LIN {X 0,Y 144.204,Z 524.14,A -85,B 0,C 180,E1 -26321.99,E2 -26321.99} C_VEL
LIN {X 0,Y 135.871,Z 530.336,A -85,B 0,C 180,E1 -26325.708,E2 -26325.708} C_VEL
LIN {X 0,Y 129.15,Z 534.492,A -85,B 0,C 180,E1 -26329.229,E2 -26329.229} C_VEL
LIN {X 0,Y 124.469,Z 537.046,A -85,B 0,C 180,E1 -26332.231,E2 -26332.231} C_VEL
LIN {X 0,Y 117.932,Z 540.01,A -85,B 0,C 180,E1 -26337.563,E2 -26337.563} C_VEL
LIN {X 0,Y 112.138,Z 541.802,A -85,B 0,C 180,E1 -26343.976,E2 -26343.976} C_VEL
LIN {X 0,Y 108.067,Z 542.166,A -85,B 0,C 180,E1 -26351.022,E2 -26351.022} C_VEL
LIN {X 0,Y 105.891,Z 541.033,A -85,B 0,C 180,E1 -26358.513,E2 -26358.513} C_VEL
LIN {X 0,Y 105.433,Z 538.416,A -85,B 0,C 180,E1 -26366.176,E2 -26366.176} C_VEL
LIN {X 0,Y 105.739,Z 536.5,A -85,B 0,C 180,E1 -26369.998,E2 -26369.998} C_VEL
LIN {X 0,Y 105.585,Z 532.557,A -85,B 0,C 180,E1 -26375.728,E2 -26375.728} C_VEL
LIN {X 0,Y 106.291,Z 526.365,A -85,B 0,C 180,E1 -26382.407,E2 -26382.407} C_VEL
LIN {X 0,Y 107.726,Z 519.519,A -85,B 0,C 180,E1 -26388.05,E2 -26388.05} C_VEL
LIN {X 0,Y 110.21,Z 510.988,A -85,B 0,C 180,E1 -26393.485,E2 -26393.485} C_VEL
LIN {X 0,Y 112.838,Z 502.152,A -85,B 0,C 180,E1 -26397.845,E2 -26397.845} C_VEL
LIN {X 0,Y 115.825,Z 492.148,A -85,B 0,C 180,E1 -26401.702,E2 -26401.702} C_VEL
LIN {X 0,Y 118.812,Z 482.066,A -85,B 0,C 180,E1 -26404.702,E2 -26404.702} C_VEL
LIN {X 0,Y 121.726,Z 470.618,A -85,B 0,C 180,E1 -26407.315,E2 -26407.315} C_VEL
LIN {X 0,Y 123.606,Z 461.97,A -85,B 0,C 180,E1 -26408.845,E2 -26408.845} C_VEL
LIN {X 0,Y 123.986,Z 456.45,A -85,B 0,C 180,E1 -26409.818,E2 -26409.818} C_VEL
LIN {X 0,Y 122.886,Z 447.257,A -85,B 0,C 180,E1 -26411.482,E2 -26411.482} C_VEL
LIN {X 0,Y 121.565,Z 437.876,A -85,B 0,C 180,E1 -26412.9,E2 -26412.9} C_VEL
LIN {X 0,Y 121.526,Z 432.057,A -85,B 0,C 180,E1 -26413.443,E2 -26413.443} C_VEL
LIN {X 0,Y 124.402,Z 398.174,A -85,B 0,C 180,E1 -26415.575,E2 -26415.575} C_VEL
LIN {X 0,Y 123.704,Z 390.073,A -85,B 0,C 180,E1 -26416.461,E2 -26416.461} C_VEL
LIN {X 0,Y 118.365,Z 373.234,A -85,B 0,C 180,E1 -26419.573,E2 -26419.573} C_VEL
LIN {X 0,Y 113.624,Z 360.938,A -85,B 0,C 180,E1 -26422.379,E2 -26422.379} C_VEL
LIN {X 0,Y 107.274,Z 349.28,A -85,B 0,C 180,E1 -26426.161,E2 -26426.161} C_VEL
LIN {X 0,Y 104.542,Z 345.011,A -85,B 0,C 180,E1 -26427.85,E2 -26427.85} C_VEL
LIN {X 0,Y 102.828,Z 342.099,A -85,B 0,C 180,E1 -26429.006,E2 -26429.006} C_VEL
LIN {X 0,Y 101.238,Z 339.918,A -85,B 0,C 180,E1 -26430.07,E2 -26430.07} C_VEL
LIN {X 0,Y 100.677,Z 337.944,A -85,B 0,C 180,E1 -26430.606,E2 -26430.606} C_VEL
LIN {X 0,Y 100.782,Z 337.935,A -85,B 0,C 180,E1 -26435.267,E2 -26435.267} C_VEL
LIN {X 0,Y 100.814,Z 337.916,A -85,B 0,C 180,E1 -26439.601,E2 -26439.601} C_VEL
LIN {X 0,Y 101.184,Z 337.863,A -85,B 0,C 180,E1 -26447.974,E2 -26447.974} C_VEL
LIN {X 0,Y 101.264,Z 337.87,A -85,B 0,C 180,E1 -26452.022,E2 -26452.022} C_VEL
LIN {X 0,Y 101.841,Z 337.774,A -85,B 0,C 180,E1 -26460.001,E2 -26460.001} C_VEL
LIN {X 0,Y 101.237,Z 337.86,A -85,B 0,C 180,E1 -26467.982,E2 -26467.982} C_VEL
LIN {X 0,Y 101.1,Z 337.863,A -85,B 0,C 180,E1 -26473.303,E2 -26473.303} C_VEL
LIN {X 0,Y 100.812,Z 337.919,A -85,B 0,C 180,E1 -26480.401,E2 -26480.401} C_VEL
LIN {X 0,Y 100.771,Z 337.896,A -85,B 0,C 180,E1 -26484.961,E2 -26484.961} C_VEL
LIN {X 0,Y 100.685,Z 337.943,A -85,B 0,C 180,E1 -26493.115,E2 -26493.115} C_VEL
LIN {X 0,Y 100.633,Z 337.918,A -85,B 0,C 180,E1 -26499.81,E2 -26499.81} C_VEL
LIN {X 0,Y 100.639,Z 337.948,A -85,B 0,C 180,E1 -26505.71,E2 -26505.71} C_VEL
LIN {X 0,Y 100.619,Z 337.931,A -85,B 0,C 180,E1 -26511.054,E2 -26511.054} C_VEL
LIN {X 0,Y 100.687,Z 337.941,A -85,B 0,C 180,E1 -26516.89,E2 -26516.89} C_VEL
LIN {X 0,Y 100.787,Z 337.927,A -85,B 0,C 180,E1 -26525.27,E2 -26525.27} C_VEL
LIN {X 0,Y 100.805,Z 337.924,A -85,B 0,C 180,E1 -26529.601,E2 -26529.601} C_VEL
LIN {X 0,Y 101.125,Z 337.885,A -85,B 0,C 180,E1 -26537.331,E2 -26537.331} C_VEL
LIN {X 0,Y 102.17,Z 340.771,A -85,B 0,C 180,E1 -26538.28,E2 -26538.28} C_VEL
LIN {X 0,Y 104.082,Z 343.292,A -85,B 0,C 180,E1 -26539.517,E2 -26539.517} C_VEL
LIN {X 0,Y 112.366,Z 356.593,A -85,B 0,C 180,E1 -26544.485,E2 -26544.485} C_VEL
LIN {X 0,Y 119.927,Z 373.331,A -85,B 0,C 180,E1 -26548.715,E2 -26548.715} C_VEL
LIN {X 0,Y 124.992,Z 386.089,A -85,B 0,C 180,E1 -26551.329,E2 -26551.329} C_VEL
LIN {X 0,Y 121.055,Z 431.333,A -85,B 0,C 180,E1 -26554.206,E2 -26554.206} C_VEL
LIN {X 0,Y 119.221,Z 444.562,A -85,B 0,C 180,E1 -26555.591,E2 -26555.591} C_VEL
LIN {X 0,Y 116.791,Z 457.435,A -85,B 0,C 180,E1 -26557.566,E2 -26557.566} C_VEL
LIN {X 0,Y 113.893,Z 469.698,A -85,B 0,C 180,E1 -26560.203,E2 -26560.203} C_VEL
LIN {X 0,Y 110.823,Z 480.586,A -85,B 0,C 180,E1 -26563.292,E2 -26563.292} C_VEL
LIN {X 0,Y 107.694,Z 490.863,A -85,B 0,C 180,E1 -26567.078,E2 -26567.078} C_VEL
LIN {X 0,Y 104.784,Z 499.838,A -85,B 0,C 180,E1 -26571.312,E2 -26571.312} C_VEL
LIN {X 0,Y 102.059,Z 508.347,A -85,B 0,C 180,E1 -26576.462,E2 -26576.462} C_VEL
LIN {X 0,Y 99.906,Z 516.005,A -85,B 0,C 180,E1 -26582.416,E2 -26582.416} C_VEL
LIN {X 0,Y 98.446,Z 521.87,A -85,B 0,C 180,E1 -26588.251,E2 -26588.251} C_VEL
LIN {X 0,Y 97.658,Z 526.395,A -85,B 0,C 180,E1 -26593.972,E2 -26593.972} C_VEL
LIN {X 0,Y 97.689,Z 529.93,A -85,B 0,C 180,E1 -26599.646,E2 -26599.646} C_VEL
LIN {X 0,Y 98.406,Z 532.573,A -85,B 0,C 180,E1 -26605.154,E2 -26605.154} C_VEL
LIN {X 0,Y 99.872,Z 534.421,A -85,B 0,C 180,E1 -26610.488,E2 -26610.488} C_VEL
LIN {X 0,Y 102.065,Z 535.611,A -85,B 0,C 180,E1 -26615.596,E2 -26615.596} C_VEL
LIN {X 0,Y 104.928,Z 536.153,A -85,B 0,C 180,E1 -26620.433,E2 -26620.433} C_VEL
LIN {X 0,Y 108.909,Z 535.995,A -85,B 0,C 180,E1 -26625.465,E2 -26625.465} C_VEL
LIN {X 0,Y 114.037,Z 534.986,A -85,B 0,C 180,E1 -26630.435,E2 -26630.435} C_VEL
LIN {X 0,Y 119.949,Z 533.081,A -85,B 0,C 180,E1 -26634.927,E2 -26634.927} C_VEL
LIN {X 0,Y 128.424,Z 529.271,A -85,B 0,C 180,E1 -26639.999,E2 -26639.999} C_VEL
LIN {X 0,Y 136.2,Z 524.843,A -85,B 0,C 180,E1 -26643.698,E2 -26643.698} C_VEL
LIN {X 0,Y 144.662,Z 519.043,A -85,B 0,C 180,E1 -26646.994,E2 -26646.994} C_VEL
LIN {X 0,Y 152.275,Z 512.818,A -85,B 0,C 180,E1 -26649.517,E2 -26649.517} C_VEL
LIN {X 0,Y 160.205,Z 505.173,A -85,B 0,C 180,E1 -26651.777,E2 -26651.777} C_VEL
LIN {X 0,Y 168.345,Z 495.926,A -85,B 0,C 180,E1 -26653.794,E2 -26653.794} C_VEL
LIN {X 0,Y 175.893,Z 485.667,A -85,B 0,C 180,E1 -26655.433,E2 -26655.433} C_VEL
LIN {X 0,Y 182.758,Z 474.132,A -85,B 0,C 180,E1 -26656.795,E2 -26656.795} C_VEL
LIN {X 0,Y 188.597,Z 461.804,A -85,B 0,C 180,E1 -26657.91,E2 -26657.91} C_VEL
LIN {X 0,Y 192.89,Z 449.978,A -85,B 0,C 180,E1 -26658.678,E2 -26658.678} C_VEL
LIN {X 0,Y 195.848,Z 439.157,A -85,B 0,C 180,E1 -26659.203,E2 -26659.203} C_VEL
LIN {X 0,Y 195.57,Z 437.962,A -85,B 0,C 180,E1 -26662.113,E2 -26662.113} C_VEL
LIN {X 0,Y 195.496,Z 438.41,A -85,B 0,C 180,E1 -26664.285,E2 -26664.285} C_VEL
LIN {X 0,Y 195.538,Z 441.194,A -85,B 0,C 180,E1 -26667.429,E2 -26667.429} C_VEL
LIN {X 0,Y 191.453,Z 455.147,A -85,B 0,C 180,E1 -26667.987,E2 -26667.987} C_VEL
LIN {X 0,Y 186.227,Z 468.207,A -85,B 0,C 180,E1 -26668.756,E2 -26668.756} C_VEL
LIN {X 0,Y 180.077,Z 480.052,A -85,B 0,C 180,E1 -26669.729,E2 -26669.729} C_VEL
LIN {X 0,Y 173.13,Z 490.968,A -85,B 0,C 180,E1 -26670.956,E2 -26670.956} C_VEL
LIN {X 0,Y 166.328,Z 499.92,A -85,B 0,C 180,E1 -26672.318,E2 -26672.318} C_VEL
LIN {X 0,Y 157.53,Z 509.729,A -85,B 0,C 180,E1 -26674.374,E2 -26674.374} C_VEL
LIN {X 0,Y 149.078,Z 517.709,A -85,B 0,C 180,E1 -26676.731,E2 -26676.731} C_VEL
LIN {X 0,Y 140.938,Z 524.241,A -85,B 0,C 180,E1 -26679.381,E2 -26679.381} C_VEL
LIN {X 0,Y 133.327,Z 529.522,A -85,B 0,C 180,E1 -26682.439,E2 -26682.439} C_VEL
LIN {X 0,Y 126.142,Z 533.783,A -85,B 0,C 180,E1 -26685.856,E2 -26685.856} C_VEL
LIN {X 0,Y 118.487,Z 537.566,A -85,B 0,C 180,E1 -26690.451,E2 -26690.451} C_VEL
LIN {X 0,Y 112.005,Z 540.093,A -85,B 0,C 180,E1 -26695.615,E2 -26695.615} C_VEL
LIN {X 0,Y 105.797,Z 541.664,A -85,B 0,C 180,E1 -26702.287,E2 -26702.287} C_VEL
LIN {X 0,Y 101.349,Z 541.752,A -85,B 0,C 180,E1 -26709.711,E2 -26709.711} C_VEL
LIN {X 0,Y 98.949,Z 540.44,A -85,B 0,C 180,E1 -26717.695,E2 -26717.695} C_VEL
LIN {X 0,Y 98.445,Z 539.235,A -85,B 0,C 180,E1 -26721.789,E2 -26721.789} C_VEL
LIN {X 0,Y 98.499,Z 536.938,A -85,B 0,C 180,E1 -26727.315,E2 -26727.315} C_VEL
LIN {X 0,Y 98.683,Z 535.535,A -85,B 0,C 180,E1 -26729.998,E2 -26729.998} C_VEL
LIN {X 0,Y 98.543,Z 531.382,A -85,B 0,C 180,E1 -26736.139,E2 -26736.139} C_VEL
LIN {X 0,Y 99.189,Z 525.985,A -85,B 0,C 180,E1 -26742.27,E2 -26742.27} C_VEL
LIN {X 0,Y 100.645,Z 519.146,A -85,B 0,C 180,E1 -26748.312,E2 -26748.312} C_VEL
LIN {X 0,Y 103.205,Z 510.618,A -85,B 0,C 180,E1 -26754.113,E2 -26754.113} C_VEL
LIN {X 0,Y 105.951,Z 501.798,A -85,B 0,C 180,E1 -26758.742,E2 -26758.742} C_VEL
LIN {X 0,Y 109.22,Z 491.411,A -85,B 0,C 180,E1 -26762.954,E2 -26762.954} C_VEL
LIN {X 0,Y 112.206,Z 481.72,A -85,B 0,C 180,E1 -26765.956,E2 -26765.956} C_VEL
LIN {X 0,Y 115.243,Z 470.241,A -85,B 0,C 180,E1 -26768.686,E2 -26768.686} C_VEL
LIN {X 0,Y 118.067,Z 457.449,A -85,B 0,C 180,E1 -26770.9,E2 -26770.9} C_VEL
LIN {X 0,Y 120.301,Z 444.156,A -85,B 0,C 180,E1 -26772.489,E2 -26772.489} C_VEL
LIN {X 0,Y 121.526,Z 432.057,A -85,B 0,C 180,E1 -26773.443,E2 -26773.443} C_VEL
LIN {X 0,Y 121.435,Z 426.244,A -85,B 0,C 180,E1 -26773.965,E2 -26773.965} C_VEL
LIN {X 0,Y 118.145,Z 407.407,A -85,B 0,C 180,E1 -26776.532,E2 -26776.532} C_VEL
LIN {X 0,Y 118.126,Z 401.597,A -85,B 0,C 180,E1 -26777.059,E2 -26777.059} C_VEL
LIN {X 0,Y 118.078,Z 394.458,A -85,B 0,C 180,E1 -26777.721,E2 -26777.721} C_VEL
LIN {X 0,Y 117.409,Z 390.896,A -85,B 0,C 180,E1 -26778.246,E2 -26778.246} C_VEL
LIN {X 0,Y 112.107,Z 374.256,A -85,B 0,C 180,E1 -26781.6,E2 -26781.6} C_VEL
LIN {X 0,Y 108.138,Z 364.014,A -85,B 0,C 180,E1 -26784.203,E2 -26784.203} C_VEL
LIN {X 0,Y 101.886,Z 352.501,A -85,B 0,C 180,E1 -26788.245,E2 -26788.245} C_VEL
LIN {X 0,Y 98.227,Z 346.757,A -85,B 0,C 180,E1 -26790.829,E2 -26790.829} C_VEL
LIN {X 0,Y 96.222,Z 343.476,A -85,B 0,C 180,E1 -26792.398,E2 -26792.398} C_VEL
LIN {X 0,Y 94.338,Z 341.074,A -85,B 0,C 180,E1 -26793.879,E2 -26793.879} C_VEL
LIN {X 0,Y 93.705,Z 338.814,A -85,B 0,C 180,E1 -26794.634,E2 -26794.634} C_VEL
LIN {X 0,Y 93.789,Z 338.802,A -85,B 0,C 180,E1 -26802.559,E2 -26802.559} C_VEL
LIN {X 0,Y 94.088,Z 338.749,A -85,B 0,C 180,E1 -26807.052,E2 -26807.052} C_VEL
LIN {X 0,Y 94.197,Z 338.747,A -85,B 0,C 180,E1 -26811.419,E2 -26811.419} C_VEL
LIN {X 0,Y 94.77,Z 338.654,A -85,B 0,C 180,E1 -26820.001,E2 -26820.001} C_VEL
LIN {X 0,Y 94.171,Z 338.734,A -85,B 0,C 180,E1 -26828.585,E2 -26828.585} C_VEL
LIN {X 0,Y 94.02,Z 338.745,A -85,B 0,C 180,E1 -26833.663,E2 -26833.663} C_VEL
LIN {X 0,Y 93.689,Z 338.797,A -85,B 0,C 180,E1 -26842.03,E2 -26842.03} C_VEL
LIN {X 0,Y 93.616,Z 338.789,A -85,B 0,C 180,E1 -26846.773,E2 -26846.773} C_VEL
LIN {X 0,Y 93.582,Z 338.826,A -85,B 0,C 180,E1 -26854.305,E2 -26854.305} C_VEL
LIN {X 0,Y 93.526,Z 338.814,A -85,B 0,C 180,E1 -26862.557,E2 -26862.557} C_VEL
LIN {X 0,Y 93.529,Z 338.829,A -85,B 0,C 180,E1 -26868.716,E2 -26868.716} C_VEL
LIN {X 0,Y 93.583,Z 338.819,A -85,B 0,C 180,E1 -26875.702,E2 -26875.702} C_VEL
LIN {X 0,Y 93.668,Z 338.816,A -85,B 0,C 180,E1 -26884.209,E2 -26884.209} C_VEL
LIN {X 0,Y 93.687,Z 338.814,A -85,B 0,C 180,E1 -26887.974,E2 -26887.974} C_VEL
LIN {X 0,Y 93.799,Z 338.942,A -85,B 0,C 180,E1 -26893.278,E2 -26893.278} C_VEL
LIN {X 0,Y 94.891,Z 341.725,A -85,B 0,C 180,E1 -26894.334,E2 -26894.334} C_VEL
LIN {X 0,Y 97.123,Z 344.099,A -85,B 0,C 180,E1 -26895.967,E2 -26895.967} C_VEL
LIN {X 0,Y 99.179,Z 347.343,A -85,B 0,C 180,E1 -26897.528,E2 -26897.528} C_VEL
LIN {X 0,Y 107.498,Z 360.915,A -85,B 0,C 180,E1 -26902.987,E2 -26902.987} C_VEL
LIN {X 0,Y 114.636,Z 377.165,A -85,B 0,C 180,E1 -26907.352,E2 -26907.352} C_VEL
LIN {X 0,Y 118.889,Z 388.434,A -85,B 0,C 180,E1 -26909.767,E2 -26909.767} C_VEL
LIN {X 0,Y 114.656,Z 432.343,A -85,B 0,C 180,E1 -26912.641,E2 -26912.641} C_VEL
LIN {X 0,Y 112.746,Z 445.688,A -85,B 0,C 180,E1 -26914.15,E2 -26914.15} C_VEL
LIN {X 0,Y 110.205,Z 458.188,A -85,B 0,C 180,E1 -26916.178,E2 -26916.178} C_VEL
LIN {X 0,Y 107.152,Z 470.365,A -85,B 0,C 180,E1 -26918.945,E2 -26918.945} C_VEL
LIN {X 0,Y 104.007,Z 481.143,A -85,B 0,C 180,E1 -26922.192,E2 -26922.192} C_VEL
LIN {X 0,Y 100.671,Z 491.438,A -85,B 0,C 180,E1 -26926.218,E2 -26926.218} C_VEL
LIN {X 0,Y 97.377,Z 501.07,A -85,B 0,C 180,E1 -26931.156,E2 -26931.156} C_VEL
LIN {X 0,Y 94.561,Z 509.672,A -85,B 0,C 180,E1 -26936.887,E2 -26936.887} C_VEL
LIN {X 0,Y 92.485,Z 517.112,A -85,B 0,C 180,E1 -26943.288,E2 -26943.288} C_VEL
LIN {X 0,Y 91.086,Z 522.715,A -85,B 0,C 180,E1 -26949.502,E2 -26949.502} C_VEL
LIN {X 0,Y 90.487,Z 527.069,A -85,B 0,C 180,E1 -26955.65,E2 -26955.65} C_VEL
LIN {X 0,Y 90.756,Z 530.464,A -85,B 0,C 180,E1 -26961.718,E2 -26961.718} C_VEL
LIN {X 0,Y 91.8,Z 533.031,A -85,B 0,C 180,E1 -26967.593,E2 -26967.593} C_VEL
LIN {X 0,Y 93.916,Z 535.029,A -85,B 0,C 180,E1 -26973.9,E2 -26973.9} C_VEL
LIN {X 0,Y 97.161,Z 536.19,A -85,B 0,C 180,E1 -26980.113,E2 -26980.113} C_VEL
LIN {X 0,Y 101.446,Z 536.477,A -85,B 0,C 180,E1 -26985.914,E2 -26985.914} C_VEL
LIN {X 0,Y 108.249,Z 535.606,A -85,B 0,C 180,E1 -26992.538,E2 -26992.538} C_VEL
LIN {X 0,Y 116.34,Z 533.242,A -85,B 0,C 180,E1 -26998.268,E2 -26998.268} C_VEL
LIN {X 0,Y 125.407,Z 529.439,A -85,B 0,C 180,E1 -27003.212,E2 -27003.212} C_VEL
LIN {X 0,Y 134.561,Z 524.463,A -85,B 0,C 180,E1 -27007.078,E2 -27007.078} C_VEL
LIN {X 0,Y 144.5,Z 517.663,A -85,B 0,C 180,E1 -27010.519,E2 -27010.519} C_VEL
LIN {X 0,Y 153.935,Z 509.908,A -85,B 0,C 180,E1 -27013.195,E2 -27013.195} C_VEL
LIN {X 0,Y 162.792,Z 501.042,A -85,B 0,C 180,E1 -27015.326,E2 -27015.326} C_VEL
LIN {X 0,Y 170.888,Z 491.294,A -85,B 0,C 180,E1 -27017.039,E2 -27017.039} C_VEL
LIN {X 0,Y 178.182,Z 480.655,A -85,B 0,C 180,E1 -27018.393,E2 -27018.393} C_VEL
LIN {X 0,Y 184.909,Z 468.504,A -85,B 0,C 180,E1 -27019.569,E2 -27019.569} C_VEL
LIN {X 0,Y 190.067,Z 456.664,A -85,B 0,C 180,E1 -27020.435,E2 -27020.435} C_VEL
LIN {X 0,Y 193.832,Z 445.249,A -85,B 0,C 180,E1 -27021.052,E2 -27021.052} C_VEL
LIN {X 0,Y 193.728,Z 445.121,A -85,B 0,C 180,E1 -27023.844,E2 -27023.844} C_VEL
LIN {X 0,Y 193.618,Z 445.986,A -85,B 0,C 180,E1 -27024.842,E2 -27024.842} C_VEL
LIN {X 0,Y 193.316,Z 447.422,A -85,B 0,C 180,E1 -27025.56,E2 -27025.56} C_VEL
LIN {X 0,Y 188.554,Z 460.936,A -85,B 0,C 180,E1 -27026.137,E2 -27026.137} C_VEL
LIN {X 0,Y 183.163,Z 472.612,A -85,B 0,C 180,E1 -27026.859,E2 -27026.859} C_VEL
LIN {X 0,Y 175.98,Z 484.888,A -85,B 0,C 180,E1 -27027.919,E2 -27027.919} C_VEL
LIN {X 0,Y 168.914,Z 494.863,A -85,B 0,C 180,E1 -27029.101,E2 -27029.101} C_VEL
LIN {X 0,Y 161.229,Z 503.991,A -85,B 0,C 180,E1 -27030.579,E2 -27030.579} C_VEL
LIN {X 0,Y 152.238,Z 512.942,A -85,B 0,C 180,E1 -27032.592,E2 -27032.592} C_VEL
LIN {X 0,Y 142.182,Z 521.313,A -85,B 0,C 180,E1 -27035.352,E2 -27035.352} C_VEL
LIN {X 0,Y 133.834,Z 527.14,A -85,B 0,C 180,E1 -27038.027,E2 -27038.027} C_VEL
LIN {X 0,Y 126.165,Z 531.775,A -85,B 0,C 180,E1 -27041.233,E2 -27041.233} C_VEL
LIN {X 0,Y 118.795,Z 535.449,A -85,B 0,C 180,E1 -27044.769,E2 -27044.769} C_VEL
LIN {X 0,Y 110.073,Z 538.977,A -85,B 0,C 180,E1 -27050.318,E2 -27050.318} C_VEL
LIN {X 0,Y 102.653,Z 540.981,A -85,B 0,C 180,E1 -27056.787,E2 -27056.787} C_VEL
LIN {X 0,Y 96.842,Z 541.563,A -85,B 0,C 180,E1 -27064.185,E2 -27064.185} C_VEL
LIN {X 0,Y 93.142,Z 540.758,A -85,B 0,C 180,E1 -27072.431,E2 -27072.431} C_VEL
LIN {X 0,Y 91.442,Z 538.447,A -85,B 0,C 180,E1 -27081.155,E2 -27081.155} C_VEL
LIN {X 0,Y 91.465,Z 535.97,A -85,B 0,C 180,E1 -27087.298,E2 -27087.298} C_VEL
LIN {X 0,Y 91.62,Z 534.567,A -85,B 0,C 180,E1 -27089.997,E2 -27089.997} C_VEL
LIN {X 0,Y 91.508,Z 530.203,A -85,B 0,C 180,E1 -27096.613,E2 -27096.613} C_VEL
LIN {X 0,Y 92.254,Z 524.573,A -85,B 0,C 180,E1 -27103.209,E2 -27103.209} C_VEL
LIN {X 0,Y 93.945,Z 517.428,A -85,B 0,C 180,E1 -27109.67,E2 -27109.67} C_VEL
LIN {X 0,Y 96.734,Z 508.508,A -85,B 0,C 180,E1 -27115.841,E2 -27115.841} C_VEL
LIN {X 0,Y 99.813,Z 499.356,A -85,B 0,C 180,E1 -27120.693,E2 -27120.693} C_VEL
LIN {X 0,Y 103.114,Z 489.17,A -85,B 0,C 180,E1 -27124.82,E2 -27124.82} C_VEL
LIN {X 0,Y 106.506,Z 478.089,A -85,B 0,C 180,E1 -27128.213,E2 -27128.213} C_VEL
LIN {X 0,Y 109.811,Z 465.827,A -85,B 0,C 180,E1 -27130.993,E2 -27130.993} C_VEL
LIN {X 0,Y 112.552,Z 452.867,A -85,B 0,C 180,E1 -27133.072,E2 -27133.072} C_VEL
LIN {X 0,Y 114.61,Z 439.454,A -85,B 0,C 180,E1 -27134.533,E2 -27134.533} C_VEL
LIN {X 0,Y 118.126,Z 401.597,A -85,B 0,C 180,E1 -27137.059,E2 -27137.059} C_VEL
LIN {X 0,Y 117.964,Z 397.831,A -85,B 0,C 180,E1 -27137.448,E2 -27137.448} C_VEL
LIN {X 0,Y 116.248,Z 392.613,A -85,B 0,C 180,E1 -27138.445,E2 -27138.445} C_VEL
LIN {X 0,Y 113.551,Z 387.978,A -85,B 0,C 180,E1 -27139.752,E2 -27139.752} C_VEL
LIN {X 0,Y 107.478,Z 378.762,A -85,B 0,C 180,E1 -27142.894,E2 -27142.894} C_VEL
LIN {X 0,Y 105.996,Z 375.313,A -85,B 0,C 180,E1 -27143.868,E2 -27143.868} C_VEL
LIN {X 0,Y 102.793,Z 367.271,A -85,B 0,C 180,E1 -27146.108,E2 -27146.108} C_VEL
LIN {X 0,Y 96.744,Z 355.991,A -85,B 0,C 180,E1 -27150.471,E2 -27150.471} C_VEL
LIN {X 0,Y 91.925,Z 348.444,A -85,B 0,C 180,E1 -27154.357,E2 -27154.357} C_VEL
LIN {X 0,Y 89.926,Z 345.331,A -85,B 0,C 180,E1 -27156.13,E2 -27156.13} C_VEL
LIN {X 0,Y 89.388,Z 344.47,A -85,B 0,C 180,E1 -27156.634,E2 -27156.634} C_VEL
LIN {X 0,Y 87.39,Z 342.104,A -85,B 0,C 180,E1 -27158.475,E2 -27158.475} C_VEL
LIN {X 0,Y 86.629,Z 339.682,A -85,B 0,C 180,E1 -27159.522,E2 -27159.522} C_VEL
LIN {X 0,Y 86.965,Z 339.641,A -85,B 0,C 180,E1 -27165.97,E2 -27165.97} C_VEL
LIN {X 0,Y 87.105,Z 339.625,A -85,B 0,C 180,E1 -27170.715,E2 -27170.715} C_VEL
LIN {X 0,Y 87.699,Z 339.534,A -85,B 0,C 180,E1 -27180.001,E2 -27180.001} C_VEL
LIN {X 0,Y 87.08,Z 339.61,A -85,B 0,C 180,E1 -27189.29,E2 -27189.29} C_VEL
LIN {X 0,Y 86.927,Z 339.63,A -85,B 0,C 180,E1 -27194.038,E2 -27194.038} C_VEL
LIN {X 0,Y 86.658,Z 339.685,A -85,B 0,C 180,E1 -27198.931,E2 -27198.931} C_VEL
LIN {X 0,Y 86.579,Z 339.664,A -85,B 0,C 180,E1 -27206.765,E2 -27206.765} C_VEL
LIN {X 0,Y 86.5,Z 339.701,A -85,B 0,C 180,E1 -27215.666,E2 -27215.666} C_VEL
LIN {X 0,Y 86.47,Z 339.695,A -85,B 0,C 180,E1 -27222.993,E2 -27222.993} C_VEL
LIN {X 0,Y 86.451,Z 339.705,A -85,B 0,C 180,E1 -27229.436,E2 -27229.436} C_VEL
LIN {X 0,Y 86.526,Z 339.693,A -85,B 0,C 180,E1 -27235.353,E2 -27235.353} C_VEL
LIN {X 0,Y 86.583,Z 339.701,A -85,B 0,C 180,E1 -27243.241,E2 -27243.241} C_VEL
LIN {X 0,Y 86.674,Z 339.889,A -85,B 0,C 180,E1 -27248.371,E2 -27248.371} C_VEL
LIN {X 0,Y 87.661,Z 342.634,A -85,B 0,C 180,E1 -27249.596,E2 -27249.596} C_VEL
LIN {X 0,Y 90.068,Z 345.258,A -85,B 0,C 180,E1 -27251.75,E2 -27251.75} C_VEL
LIN {X 0,Y 92.267,Z 348.549,A -85,B 0,C 180,E1 -27253.677,E2 -27253.677} C_VEL
LIN {X 0,Y 93.542,Z 350.242,A -85,B 0,C 180,E1 -27254.696,E2 -27254.696} C_VEL
LIN {X 0,Y 97.922,Z 357.186,A -85,B 0,C 180,E1 -27258.097,E2 -27258.097} C_VEL
LIN {X 0,Y 102.763,Z 365.554,A -85,B 0,C 180,E1 -27261.474,E2 -27261.474} C_VEL
LIN {X 0,Y 109.271,Z 380.585,A -85,B 0,C 180,E1 -27265.764,E2 -27265.764} C_VEL
LIN {X 0,Y 112.743,Z 390.161,A -85,B 0,C 180,E1 -27267.97,E2 -27267.97} C_VEL
LIN {X 0,Y 108.502,Z 432.395,A -85,B 0,C 180,E1 -27270.827,E2 -27270.827} C_VEL
LIN {X 0,Y 106.496,Z 445.811,A -85,B 0,C 180,E1 -27272.393,E2 -27272.393} C_VEL
LIN {X 0,Y 103.662,Z 458.967,A -85,B 0,C 180,E1 -27274.62,E2 -27274.62} C_VEL
LIN {X 0,Y 100.426,Z 471.127,A -85,B 0,C 180,E1 -27277.542,E2 -27277.542} C_VEL
LIN {X 0,Y 97.166,Z 481.854,A -85,B 0,C 180,E1 -27280.988,E2 -27280.988} C_VEL
LIN {X 0,Y 93.526,Z 492.396,A -85,B 0,C 180,E1 -27285.42,E2 -27285.42} C_VEL
LIN {X 0,Y 90.159,Z 501.831,A -85,B 0,C 180,E1 -27290.7,E2 -27290.7} C_VEL
LIN {X 0,Y 87.088,Z 510.956,A -85,B 0,C 180,E1 -27297.412,E2 -27297.412} C_VEL
LIN {X 0,Y 85.058,Z 518.053,A -85,B 0,C 180,E1 -27304.281,E2 -27304.281} C_VEL
LIN {X 0,Y 83.651,Z 524.325,A -85,B 0,C 180,E1 -27312.235,E2 -27312.235} C_VEL
LIN {X 0,Y 83.496,Z 528.602,A -85,B 0,C 180,E1 -27319.252,E2 -27319.252} C_VEL
LIN {X 0,Y 84.357,Z 531.99,A -85,B 0,C 180,E1 -27326.426,E2 -27326.426} C_VEL
LIN {X 0,Y 86.418,Z 534.461,A -85,B 0,C 180,E1 -27333.46,E2 -27333.46} C_VEL
LIN {X 0,Y 90.718,Z 536.311,A -85,B 0,C 180,E1 -27341.947,E2 -27341.947} C_VEL
LIN {X 0,Y 94.561,Z 536.8,A -85,B 0,C 180,E1 -27347.115,E2 -27347.115} C_VEL
LIN {X 0,Y 99.349,Z 536.592,A -85,B 0,C 180,E1 -27352.054,E2 -27352.054} C_VEL
LIN {X 0,Y 105.563,Z 535.568,A -85,B 0,C 180,E1 -27357.054,E2 -27357.054} C_VEL
LIN {X 0,Y 112.487,Z 533.676,A -85,B 0,C 180,E1 -27361.449,E2 -27361.449} C_VEL
LIN {X 0,Y 119.993,Z 530.87,A -85,B 0,C 180,E1 -27365.304,E2 -27365.304} C_VEL
LIN {X 0,Y 129.939,Z 526.025,A -85,B 0,C 180,E1 -27369.337,E2 -27369.337} C_VEL
LIN {X 0,Y 139.209,Z 520.414,A -85,B 0,C 180,E1 -27372.39,E2 -27372.39} C_VEL
LIN {X 0,Y 148.955,Z 513.208,A -85,B 0,C 180,E1 -27375.04,E2 -27375.04} C_VEL
LIN {X 0,Y 157.383,Z 505.668,A -85,B 0,C 180,E1 -27376.997,E2 -27376.997} C_VEL
LIN {X 0,Y 166.083,Z 496.428,A -85,B 0,C 180,E1 -27378.739,E2 -27378.739} C_VEL
LIN {X 0,Y 173.909,Z 486.429,A -85,B 0,C 180,E1 -27380.118,E2 -27380.118} C_VEL
LIN {X 0,Y 180.977,Z 475.296,A -85,B 0,C 180,E1 -27381.248,E2 -27381.248} C_VEL
LIN {X 0,Y 187.076,Z 463.26,A -85,B 0,C 180,E1 -27382.189,E2 -27382.189} C_VEL
LIN {X 0,Y 191.414,Z 452.286,A -85,B 0,C 180,E1 -27382.824,E2 -27382.824} C_VEL
LIN {X 0,Y 191.621,Z 451.796,A -85,B 0,C 180,E1 -27383.519,E2 -27383.519} C_VEL
LIN {X 0,Y 189.954,Z 456.449,A -85,B 0,C 180,E1 -27383.769,E2 -27383.769} C_VEL
LIN {X 0,Y 184.28,Z 469.374,A -85,B 0,C 180,E1 -27384.418,E2 -27384.418} C_VEL
LIN {X 0,Y 177.751,Z 481.044,A -85,B 0,C 180,E1 -27385.25,E2 -27385.25} C_VEL
LIN {X 0,Y 170.452,Z 491.649,A -85,B 0,C 180,E1 -27386.259,E2 -27386.259} C_VEL
LIN {X 0,Y 162.504,Z 501.193,A -85,B 0,C 180,E1 -27387.55,E2 -27387.55} C_VEL
LIN {X 0,Y 153.193,Z 510.603,A -85,B 0,C 180,E1 -27389.346,E2 -27389.346} C_VEL
LIN {X 0,Y 144.133,Z 518.297,A -85,B 0,C 180,E1 -27391.424,E2 -27391.424} C_VEL
LIN {X 0,Y 135.345,Z 524.573,A -85,B 0,C 180,E1 -27393.814,E2 -27393.814} C_VEL
LIN {X 0,Y 126.952,Z 529.643,A -85,B 0,C 180,E1 -27396.607,E2 -27396.607} C_VEL
LIN {X 0,Y 118.986,Z 533.714,A -85,B 0,C 180,E1 -27399.836,E2 -27399.836} C_VEL
LIN {X 0,Y 113.931,Z 535.924,A -85,B 0,C 180,E1 -27402.246,E2 -27402.246} C_VEL
LIN {X 0,Y 104.697,Z 539.109,A -85,B 0,C 180,E1 -27407.832,E2 -27407.832} C_VEL
LIN {X 0,Y 96.782,Z 540.87,A -85,B 0,C 180,E1 -27414.481,E2 -27414.481} C_VEL
LIN {X 0,Y 90.503,Z 541.233,A -85,B 0,C 180,E1 -27422.227,E2 -27422.227} C_VEL
LIN {X 0,Y 86.401,Z 540.157,A -85,B 0,C 180,E1 -27431.009,E2 -27431.009} C_VEL
LIN {X 0,Y 84.463,Z 537.633,A -85,B 0,C 180,E1 -27440.418,E2 -27440.418} C_VEL
LIN {X 0,Y 84.445,Z 534.955,A -85,B 0,C 180,E1 -27447.074,E2 -27447.074} C_VEL
LIN {X 0,Y 84.572,Z 533.499,A -85,B 0,C 180,E1 -27449.997,E2 -27449.997} C_VEL
LIN {X 0,Y 84.501,Z 528.93,A -85,B 0,C 180,E1 -27457.164,E2 -27457.164} C_VEL
LIN {X 0,Y 85.361,Z 523.043,A -85,B 0,C 180,E1 -27464.297,E2 -27464.297} C_VEL
LIN {X 0,Y 87.312,Z 515.636,A -85,B 0,C 180,E1 -27471.233,E2 -27471.233} C_VEL
LIN {X 0,Y 89.803,Z 508.043,A -85,B 0,C 180,E1 -27476.74,E2 -27476.74} C_VEL
LIN {X 0,Y 93.055,Z 498.854,A -85,B 0,C 180,E1 -27481.913,E2 -27481.913} C_VEL
LIN {X 0,Y 96.667,Z 488.209,A -85,B 0,C 180,E1 -27486.424,E2 -27486.424} C_VEL
LIN {X 0,Y 100.088,Z 477.462,A -85,B 0,C 180,E1 -27489.844,E2 -27489.844} C_VEL
LIN {X 0,Y 103.531,Z 465.057,A -85,B 0,C 180,E1 -27492.749,E2 -27492.749} C_VEL
LIN {X 0,Y 106.43,Z 451.978,A -85,B 0,C 180,E1 -27494.886,E2 -27494.886} C_VEL
LIN {X 0,Y 108.481,Z 438.789,A -85,B 0,C 180,E1 -27496.355,E2 -27496.355} C_VEL
LIN {X 0,Y 112.186,Z 399.571,A -85,B 0,C 180,E1 -27499.079,E2 -27499.079} C_VEL
LIN {X 0,Y 111.775,Z 393.986,A -85,B 0,C 180,E1 -27499.764,E2 -27499.764} C_VEL
LIN {X 0,Y 106.706,Z 377.419,A -85,B 0,C 180,E1 -27503.347,E2 -27503.347} C_VEL
LIN {X 0,Y 105.996,Z 375.313,A -85,B 0,C 180,E1 -27503.868,E2 -27503.868} C_VEL
LIN {X 0,Y 104.266,Z 372.364,A -85,B 0,C 180,E1 -27504.916,E2 -27504.916} C_VEL
LIN {X 0,Y 100.088,Z 369.012,A -85,B 0,C 180,E1 -27507.165,E2 -27507.165} C_VEL
LIN {X 0,Y 95.783,Z 365.906,A -85,B 0,C 180,E1 -27509.714,E2 -27509.714} C_VEL
LIN {X 0,Y 93.827,Z 363.274,A -85,B 0,C 180,E1 -27511.156,E2 -27511.156} C_VEL
LIN {X 0,Y 88.432,Z 354.194,A -85,B 0,C 180,E1 -27515.821,E2 -27515.821} C_VEL
LIN {X 0,Y 85.433,Z 349.742,A -85,B 0,C 180,E1 -27518.749,E2 -27518.749} C_VEL
LIN {X 0,Y 83.202,Z 346.241,A -85,B 0,C 180,E1 -27521.215,E2 -27521.215} C_VEL
LIN {X 0,Y 82.229,Z 345.221,A -85,B 0,C 180,E1 -27522.274,E2 -27522.274} C_VEL
LIN {X 0,Y 80.42,Z 342.811,A -85,B 0,C 180,E1 -27524.477,E2 -27524.477} C_VEL
LIN {X 0,Y 79.837,Z 340.531,A -85,B 0,C 180,E1 -27525.527,E2 -27525.527} C_VEL
LIN {X 0,Y 79.99,Z 340.505,A -85,B 0,C 180,E1 -27529.88,E2 -27529.88} C_VEL
LIN {X 0,Y 80.628,Z 340.414,A -85,B 0,C 180,E1 -27540.001,E2 -27540.001} C_VEL
LIN {X 0,Y 79.963,Z 340.49,A -85,B 0,C 180,E1 -27550.125,E2 -27550.125} C_VEL
LIN {X 0,Y 79.744,Z 340.534,A -85,B 0,C 180,E1 -27555.332,E2 -27555.332} C_VEL
LIN {X 0,Y 79.518,Z 340.568,A -85,B 0,C 180,E1 -27560.705,E2 -27560.705} C_VEL
LIN {X 0,Y 79.477,Z 340.553,A -85,B 0,C 180,E1 -27567.844,E2 -27567.844} C_VEL
LIN {X 0,Y 79.372,Z 340.597,A -85,B 0,C 180,E1 -27572.093,E2 -27572.093} C_VEL
LIN {X 0,Y 79.36,Z 340.569,A -85,B 0,C 180,E1 -27578.311,E2 -27578.311} C_VEL
LIN {X 0,Y 79.383,Z 340.593,A -85,B 0,C 180,E1 -27585.096,E2 -27585.096} C_VEL
LIN {X 0,Y 79.382,Z 340.57,A -85,B 0,C 180,E1 -27592.829,E2 -27592.829} C_VEL
LIN {X 0,Y 79.492,Z 340.772,A -85,B 0,C 180,E1 -27601.987,E2 -27601.987} C_VEL
LIN {X 0,Y 80.585,Z 343.489,A -85,B 0,C 180,E1 -27603.639,E2 -27603.639} C_VEL
LIN {X 0,Y 82.632,Z 345.596,A -85,B 0,C 180,E1 -27605.927,E2 -27605.927} C_VEL
LIN {X 0,Y 83.234,Z 346.298,A -85,B 0,C 180,E1 -27606.582,E2 -27606.582} C_VEL
LIN {X 0,Y 85.226,Z 349.532,A -85,B 0,C 180,E1 -27608.826,E2 -27608.826} C_VEL
LIN {X 0,Y 86.53,Z 351.079,A -85,B 0,C 180,E1 -27610.102,E2 -27610.102} C_VEL
LIN {X 0,Y 90.588,Z 357.015,A -85,B 0,C 180,E1 -27613.829,E2 -27613.829} C_VEL
LIN {X 0,Y 96.554,Z 367.185,A -85,B 0,C 180,E1 -27618.645,E2 -27618.645} C_VEL
LIN {X 0,Y 98.534,Z 371.14,A -85,B 0,C 180,E1 -27620.147,E2 -27620.147} C_VEL
LIN {X 0,Y 104.014,Z 384.27,A -85,B 0,C 180,E1 -27624.105,E2 -27624.105} C_VEL
LIN {X 0,Y 106.742,Z 391.868,A -85,B 0,C 180,E1 -27625.977,E2 -27625.977} C_VEL
LIN {X 0,Y 102.499,Z 432.209,A -85,B 0,C 180,E1 -27628.789,E2 -27628.789} C_VEL
LIN {X 0,Y 100.399,Z 445.541,A -85,B 0,C 180,E1 -27630.378,E2 -27630.378} C_VEL
LIN {X 0,Y 97.614,Z 458.085,A -85,B 0,C 180,E1 -27632.546,E2 -27632.546} C_VEL
LIN {X 0,Y 94.153,Z 470.611,A -85,B 0,C 180,E1 -27635.625,E2 -27635.625} C_VEL
LIN {X 0,Y 90.463,Z 482.129,A -85,B 0,C 180,E1 -27639.505,E2 -27639.505} C_VEL
LIN {X 0,Y 86.711,Z 492.37,A -85,B 0,C 180,E1 -27644.075,E2 -27644.075} C_VEL
LIN {X 0,Y 83.181,Z 501.877,A -85,B 0,C 180,E1 -27649.756,E2 -27649.756} C_VEL
LIN {X 0,Y 79.973,Z 511.01,A -85,B 0,C 180,E1 -27656.99,E2 -27656.99} C_VEL
LIN {X 0,Y 77.973,Z 517.759,A -85,B 0,C 180,E1 -27663.993,E2 -27663.993} C_VEL
LIN {X 0,Y 76.535,Z 524.186,A -85,B 0,C 180,E1 -27672.722,E2 -27672.722} C_VEL
LIN {X 0,Y 76.443,Z 528.316,A -85,B 0,C 180,E1 -27679.94,E2 -27679.94} C_VEL
LIN {X 0,Y 78.068,Z 532.704,A -85,B 0,C 180,E1 -27690.154,E2 -27690.154} C_VEL
LIN {X 0,Y 82.116,Z 535.702,A -85,B 0,C 180,E1 -27700.304,E2 -27700.304} C_VEL
LIN {X 0,Y 86.537,Z 536.838,A -85,B 0,C 180,E1 -27707.059,E2 -27707.059} C_VEL
LIN {X 0,Y 92.037,Z 537.093,A -85,B 0,C 180,E1 -27713.085,E2 -27713.085} C_VEL
LIN {X 0,Y 100.795,Z 536.121,A -85,B 0,C 180,E1 -27719.999,E2 -27719.999} C_VEL
LIN {X 0,Y 106.994,Z 534.678,A -85,B 0,C 180,E1 -27723.765,E2 -27723.765} C_VEL
LIN {X 0,Y 117.181,Z 531.3,A -85,B 0,C 180,E1 -27728.623,E2 -27728.623} C_VEL
LIN {X 0,Y 124.814,Z 527.954,A -85,B 0,C 180,E1 -27731.512,E2 -27731.512} C_VEL
LIN {X 0,Y 133.005,Z 523.584,A -85,B 0,C 180,E1 -27734.095,E2 -27734.095} C_VEL
LIN {X 0,Y 141.366,Z 518.238,A -85,B 0,C 180,E1 -27736.37,E2 -27736.37} C_VEL
LIN {X 0,Y 149.984,Z 511.759,A -85,B 0,C 180,E1 -27738.344,E2 -27738.344} C_VEL
LIN {X 0,Y 158.814,Z 503.851,A -85,B 0,C 180,E1 -27740.082,E2 -27740.082} C_VEL
LIN {X 0,Y 167.081,Z 494.972,A -85,B 0,C 180,E1 -27741.514,E2 -27741.514} C_VEL
LIN {X 0,Y 175.295,Z 484.183,A -85,B 0,C 180,E1 -27742.759,E2 -27742.759} C_VEL
LIN {X 0,Y 175.742,Z 483.563,A -85,B 0,C 180,E1 -27743.104,E2 -27743.104} C_VEL
LIN {X 0,Y 167.536,Z 494.624,A -85,B 0,C 180,E1 -27744.159,E2 -27744.159} C_VEL
LIN {X 0,Y 159.444,Z 503.653,A -85,B 0,C 180,E1 -27745.362,E2 -27745.362} C_VEL
LIN {X 0,Y 149.915,Z 512.492,A -85,B 0,C 180,E1 -27747.033,E2 -27747.033} C_VEL
LIN {X 0,Y 139.092,Z 520.804,A -85,B 0,C 180,E1 -27749.352,E2 -27749.352} C_VEL
LIN {X 0,Y 128.615,Z 527.417,A -85,B 0,C 180,E1 -27752.113,E2 -27752.113} C_VEL
LIN {X 0,Y 120.085,Z 531.868,A -85,B 0,C 180,E1 -27754.977,E2 -27754.977} C_VEL
LIN {X 0,Y 109.294,Z 536.295,A -85,B 0,C 180,E1 -27759.495,E2 -27759.495} C_VEL
LIN {X 0,Y 99.533,Z 539.239,A -85,B 0,C 180,E1 -27765.079,E2 -27765.079} C_VEL
LIN {X 0,Y 91.089,Z 540.737,A -85,B 0,C 180,E1 -27771.882,E2 -27771.882} C_VEL
LIN {X 0,Y 84.288,Z 540.81,A -85,B 0,C 180,E1 -27779.978,E2 -27779.978} C_VEL
LIN {X 0,Y 79.726,Z 539.517,A -85,B 0,C 180,E1 -27789.35,E2 -27789.35} C_VEL
LIN {X 0,Y 77.509,Z 536.784,A -85,B 0,C 180,E1 -27799.549,E2 -27799.549} C_VEL
LIN {X 0,Y 77.427,Z 533.934,A -85,B 0,C 180,E1 -27806.808,E2 -27806.808} C_VEL
LIN {X 0,Y 77.52,Z 532.363,A -85,B 0,C 180,E1 -27809.997,E2 -27809.997} C_VEL
LIN {X 0,Y 77.511,Z 527.562,A -85,B 0,C 180,E1 -27817.814,E2 -27817.814} C_VEL
LIN {X 0,Y 78.516,Z 521.413,A -85,B 0,C 180,E1 -27825.574,E2 -27825.574} C_VEL
LIN {X 0,Y 80.747,Z 513.688,A -85,B 0,C 180,E1 -27833.055,E2 -27833.055} C_VEL
LIN {X 0,Y 83.537,Z 505.768,A -85,B 0,C 180,E1 -27838.927,E2 -27838.927} C_VEL
LIN {X 0,Y 87.496,Z 495.057,A -85,B 0,C 180,E1 -27844.908,E2 -27844.908} C_VEL
LIN {X 0,Y 91.038,Z 485.166,A -85,B 0,C 180,E1 -27849.014,E2 -27849.014} C_VEL
LIN {X 0,Y 94.808,Z 473.583,A -85,B 0,C 180,E1 -27852.561,E2 -27852.561} C_VEL
LIN {X 0,Y 98.173,Z 461.08,A -85,B 0,C 180,E1 -27855.346,E2 -27855.346} C_VEL
LIN {X 0,Y 100.958,Z 448.061,A -85,B 0,C 180,E1 -27857.327,E2 -27857.327} C_VEL
LIN {X 0,Y 102.909,Z 434.33,A -85,B 0,C 180,E1 -27858.693,E2 -27858.693} C_VEL
LIN {X 0,Y 106.255,Z 400.127,A -85,B 0,C 180,E1 -27861.106,E2 -27861.106} C_VEL
LIN {X 0,Y 106,Z 396.211,A -85,B 0,C 180,E1 -27861.618,E2 -27861.618} C_VEL
LIN {X 0,Y 101.058,Z 379.734,A -85,B 0,C 180,E1 -27865.444,E2 -27865.444} C_VEL
LIN {X 0,Y 97.965,Z 371.483,A -85,B 0,C 180,E1 -27867.872,E2 -27867.872} C_VEL
LIN {X 0,Y 93.827,Z 363.274,A -85,B 0,C 180,E1 -27871.156,E2 -27871.156} C_VEL
LIN {X 0,Y 91.911,Z 360.836,A -85,B 0,C 180,E1 -27872.629,E2 -27872.629} C_VEL
LIN {X 0,Y 87.78,Z 358.545,A -85,B 0,C 180,E1 -27875.626,E2 -27875.626} C_VEL
LIN {X 0,Y 82.872,Z 356.133,A -85,B 0,C 180,E1 -27879.76,E2 -27879.76} C_VEL
LIN {X 0,Y 81.578,Z 354.781,A -85,B 0,C 180,E1 -27881.133,E2 -27881.133} C_VEL
LIN {X 0,Y 79.352,Z 351.328,A -85,B 0,C 180,E1 -27883.851,E2 -27883.851} C_VEL
LIN {X 0,Y 77.237,Z 348.491,A -85,B 0,C 180,E1 -27886.633,E2 -27886.633} C_VEL
LIN {X 0,Y 76.427,Z 346.729,A -85,B 0,C 180,E1 -27887.95,E2 -27887.95} C_VEL
LIN {X 0,Y 73.921,Z 344.2,A -85,B 0,C 180,E1 -27891.802,E2 -27891.802} C_VEL
LIN {X 0,Y 73.038,Z 341.685,A -85,B 0,C 180,E1 -27893.787,E2 -27893.787} C_VEL
LIN {X 0,Y 73.039,Z 341.385,A -85,B 0,C 180,E1 -27894.133,E2 -27894.133} C_VEL
LIN {X 0,Y 73.556,Z 341.294,A -85,B 0,C 180,E1 -27900.001,E2 -27900.001} C_VEL
LIN {X 0,Y 72.854,Z 341.371,A -85,B 0,C 180,E1 -27911.125,E2 -27911.125} C_VEL
LIN {X 0,Y 72.574,Z 341.436,A -85,B 0,C 180,E1 -27916.89,E2 -27916.89} C_VEL
LIN {X 0,Y 72.394,Z 341.436,A -85,B 0,C 180,E1 -27922.851,E2 -27922.851} C_VEL
LIN {X 0,Y 72.355,Z 341.449,A -85,B 0,C 180,E1 -27929.058,E2 -27929.058} C_VEL
LIN {X 0,Y 72.289,Z 341.469,A -85,B 0,C 180,E1 -27935.687,E2 -27935.687} C_VEL
LIN {X 0,Y 72.243,Z 341.462,A -85,B 0,C 180,E1 -27942.923,E2 -27942.923} C_VEL
LIN {X 0,Y 72.29,Z 341.456,A -85,B 0,C 180,E1 -27951.058,E2 -27951.058} C_VEL
LIN {X 0,Y 72.36,Z 341.563,A -85,B 0,C 180,E1 -27952.923,E2 -27952.923} C_VEL
LIN {X 0,Y 73.002,Z 343.792,A -85,B 0,C 180,E1 -27954.523,E2 -27954.523} C_VEL
LIN {X 0,Y 74.675,Z 345.942,A -85,B 0,C 180,E1 -27957.453,E2 -27957.453} C_VEL
LIN {X 0,Y 76.522,Z 347.303,A -85,B 0,C 180,E1 -27960.088,E2 -27960.088} C_VEL
LIN {X 0,Y 78.45,Z 350.578,A -85,B 0,C 180,E1 -27962.909,E2 -27962.909} C_VEL
LIN {X 0,Y 79.951,Z 352.186,A -85,B 0,C 180,E1 -27964.709,E2 -27964.709} C_VEL
LIN {X 0,Y 82.518,Z 355.91,A -85,B 0,C 180,E1 -27967.672,E2 -27967.672} C_VEL
LIN {X 0,Y 87.047,Z 362.769,A -85,B 0,C 180,E1 -27972.329,E2 -27972.329} C_VEL
LIN {X 0,Y 93.337,Z 374.15,A -85,B 0,C 180,E1 -27977.801,E2 -27977.801} C_VEL
LIN {X 0,Y 98.742,Z 387.616,A -85,B 0,C 180,E1 -27982.229,E2 -27982.229} C_VEL
LIN {X 0,Y 100.824,Z 393.59,A -85,B 0,C 180,E1 -27983.833,E2 -27983.833} C_VEL
LIN {X 0,Y 96.372,Z 433.137,A -85,B 0,C 180,E1 -27986.671,E2 -27986.671} C_VEL
LIN {X 0,Y 94.071,Z 446.796,A -85,B 0,C 180,E1 -27988.397,E2 -27988.397} C_VEL
LIN {X 0,Y 90.907,Z 460.04,A -85,B 0,C 180,E1 -27990.876,E2 -27990.876} C_VEL
LIN {X 0,Y 87.325,Z 472.03,A -85,B 0,C 180,E1 -27994.066,E2 -27994.066} C_VEL
LIN {X 0,Y 83.594,Z 482.958,A -85,B 0,C 180,E1 -27998.03,E2 -27998.03} C_VEL
LIN {X 0,Y 79.442,Z 493.713,A -85,B 0,C 180,E1 -28003.303,E2 -28003.303} C_VEL
LIN {X 0,Y 75.637,Z 503.48,A -85,B 0,C 180,E1 -28009.813,E2 -28009.813} C_VEL
LIN {X 0,Y 72.663,Z 511.75,A -85,B 0,C 180,E1 -28017.17,E2 -28017.17} C_VEL
LIN {X 0,Y 70.618,Z 518.307,A -85,B 0,C 180,E1 -28024.818,E2 -28024.818} C_VEL
LIN {X 0,Y 69.32,Z 524.799,A -85,B 0,C 180,E1 -28034.788,E2 -28034.788} C_VEL
LIN {X 0,Y 69.716,Z 529.3,A -85,B 0,C 180,E1 -28043.757,E2 -28043.757} C_VEL
LIN {X 0,Y 71.438,Z 532.668,A -85,B 0,C 180,E1 -28052.308,E2 -28052.308} C_VEL
LIN {X 0,Y 74.605,Z 535.123,A -85,B 0,C 180,E1 -28060.403,E2 -28060.403} C_VEL
LIN {X 0,Y 80.776,Z 536.986,A -85,B 0,C 180,E1 -28069.978,E2 -28069.978} C_VEL
LIN {X 0,Y 85.793,Z 537.424,A -85,B 0,C 180,E1 -28075.3,E2 -28075.3} C_VEL
LIN {X 0,Y 91.496,Z 537.206,A -85,B 0,C 180,E1 -28079.999,E2 -28079.999} C_VEL
LIN {X 0,Y 98.723,Z 536.214,A -85,B 0,C 180,E1 -28084.67,E2 -28084.67} C_VEL
LIN {X 0,Y 106.662,Z 534.375,A -85,B 0,C 180,E1 -28088.742,E2 -28088.742} C_VEL
LIN {X 0,Y 115.047,Z 531.66,A -85,B 0,C 180,E1 -28092.194,E2 -28092.194} C_VEL
LIN {X 0,Y 123.737,Z 528.015,A -85,B 0,C 180,E1 -28095.073,E2 -28095.073} C_VEL
LIN {X 0,Y 135.194,Z 521.916,A -85,B 0,C 180,E1 -28098.174,E2 -28098.174} C_VEL
LIN {X 0,Y 145.705,Z 514.915,A -85,B 0,C 180,E1 -28100.449,E2 -28100.449} C_VEL
LIN {X 0,Y 155.386,Z 507.011,A -85,B 0,C 180,E1 -28102.224,E2 -28102.224} C_VEL
LIN {X 0,Y 156.965,Z 505.536,A -85,B 0,C 180,E1 -28102.494,E2 -28102.494} C_VEL
LIN {X 0,Y 156.613,Z 505.916,A -85,B 0,C 180,E1 -28103.08,E2 -28103.08} C_VEL
LIN {X 0,Y 146.885,Z 514.342,A -85,B 0,C 180,E1 -28104.617,E2 -28104.617} C_VEL
LIN {X 0,Y 137.381,Z 521.184,A -85,B 0,C 180,E1 -28106.457,E2 -28106.457} C_VEL
LIN {X 0,Y 128.071,Z 526.77,A -85,B 0,C 180,E1 -28108.593,E2 -28108.593} C_VEL
LIN {X 0,Y 119.083,Z 531.275,A -85,B 0,C 180,E1 -28111.153,E2 -28111.153} C_VEL
LIN {X 0,Y 110.46,Z 534.811,A -85,B 0,C 180,E1 -28114.193,E2 -28114.193} C_VEL
LIN {X 0,Y 99.637,Z 538.189,A -85,B 0,C 180,E1 -28119.11,E2 -28119.11} C_VEL
LIN {X 0,Y 89.981,Z 540.088,A -85,B 0,C 180,E1 -28125.332,E2 -28125.332} C_VEL
LIN {X 0,Y 81.71,Z 540.622,A -85,B 0,C 180,E1 -28132.978,E2 -28132.978} C_VEL
LIN {X 0,Y 75.289,Z 539.787,A -85,B 0,C 180,E1 -28142.174,E2 -28142.174} C_VEL
LIN {X 0,Y 71.542,Z 537.513,A -85,B 0,C 180,E1 -28152.857,E2 -28152.857} C_VEL
LIN {X 0,Y 70.358,Z 533.741,A -85,B 0,C 180,E1 -28164.264,E2 -28164.264} C_VEL
LIN {X 0,Y 70.471,Z 531.2,A -85,B 0,C 180,E1 -28169.997,E2 -28169.997} C_VEL
LIN {X 0,Y 70.51,Z 526.173,A -85,B 0,C 180,E1 -28178.595,E2 -28178.595} C_VEL
LIN {X 0,Y 71.726,Z 519.709,A -85,B 0,C 180,E1 -28187.091,E2 -28187.091} C_VEL
LIN {X 0,Y 74.3,Z 511.621,A -85,B 0,C 180,E1 -28195.188,E2 -28195.188} C_VEL
LIN {X 0,Y 77.402,Z 503.34,A -85,B 0,C 180,E1 -28201.469,E2 -28201.469} C_VEL
LIN {X 0,Y 81.357,Z 493.221,A -85,B 0,C 180,E1 -28207.203,E2 -28207.203} C_VEL
LIN {X 0,Y 85.674,Z 481.55,A -85,B 0,C 180,E1 -28211.984,E2 -28211.984} C_VEL
LIN {X 0,Y 89.183,Z 470.899,A -85,B 0,C 180,E1 -28215.169,E2 -28215.169} C_VEL
LIN {X 0,Y 92.477,Z 458.761,A -85,B 0,C 180,E1 -28217.81,E2 -28217.81} C_VEL
LIN {X 0,Y 95.256,Z 445.769,A -85,B 0,C 180,E1 -28219.739,E2 -28219.739} C_VEL
LIN {X 0,Y 97.003,Z 433.535,A -85,B 0,C 180,E1 -28220.945,E2 -28220.945} C_VEL
LIN {X 0,Y 100.406,Z 400.29,A -85,B 0,C 180,E1 -28223.375,E2 -28223.375} C_VEL
LIN {X 0,Y 100.091,Z 397.827,A -85,B 0,C 180,E1 -28223.786,E2 -28223.786} C_VEL
LIN {X 0,Y 95.792,Z 382.821,A -85,B 0,C 180,E1 -28227.544,E2 -28227.544} C_VEL
LIN {X 0,Y 93.102,Z 375.384,A -85,B 0,C 180,E1 -28229.936,E2 -28229.936} C_VEL
LIN {X 0,Y 87.969,Z 365.22,A -85,B 0,C 180,E1 -28234.464,E2 -28234.464} C_VEL
LIN {X 0,Y 83.952,Z 358.512,A -85,B 0,C 180,E1 -28238.456,E2 -28238.456} C_VEL
LIN {X 0,Y 81.678,Z 354.918,A -85,B 0,C 180,E1 -28241.018,E2 -28241.018} C_VEL
LIN {X 0,Y 81.578,Z 354.781,A -85,B 0,C 180,E1 -28241.133,E2 -28241.133} C_VEL
LIN {X 0,Y 78.883,Z 351.885,A -85,B 0,C 180,E1 -28244.259,E2 -28244.259} C_VEL
LIN {X 0,Y 76.011,Z 349.888,A -85,B 0,C 180,E1 -28247.802,E2 -28247.802} C_VEL
LIN {X 0,Y 67.797,Z 345.868,A -85,B 0,C 180,E1 -28262.13,E2 -28262.13} C_VEL
LIN {X 0,Y 66.02,Z 343.333,A -85,B 0,C 180,E1 -28268.418,E2 -28268.418} C_VEL
LIN {X 0,Y 65.799,Z 342.252,A -85,B 0,C 180,E1 -28269.997,E2 -28269.997} C_VEL
LIN {X 0,Y 65.616,Z 342.29,A -85,B 0,C 180,E1 -28275.441,E2 -28275.441} C_VEL
LIN {X 0,Y 65.228,Z 342.318,A -85,B 0,C 180,E1 -28285.532,E2 -28285.532} C_VEL
LIN {X 0,Y 65.166,Z 342.368,A -85,B 0,C 180,E1 -28292.634,E2 -28292.634} C_VEL
LIN {X 0,Y 65.265,Z 342.479,A -85,B 0,C 180,E1 -28295.962,E2 -28295.962} C_VEL
LIN {X 0,Y 66.283,Z 345.341,A -85,B 0,C 180,E1 -28301.305,E2 -28301.305} C_VEL
LIN {X 0,Y 68.944,Z 347.77,A -85,B 0,C 180,E1 -28308.862,E2 -28308.862} C_VEL
LIN {X 0,Y 69.883,Z 348.39,A -85,B 0,C 180,E1 -28310.835,E2 -28310.835} C_VEL
LIN {X 0,Y 71.417,Z 351.336,A -85,B 0,C 180,E1 -28314.219,E2 -28314.219} C_VEL
LIN {X 0,Y 73.852,Z 353.709,A -85,B 0,C 180,E1 -28318.282,E2 -28318.282} C_VEL
LIN {X 0,Y 76.06,Z 357.125,A -85,B 0,C 180,E1 -28321.729,E2 -28321.729} C_VEL
LIN {X 0,Y 77.418,Z 359.16,A -85,B 0,C 180,E1 -28323.602,E2 -28323.602} C_VEL
LIN {X 0,Y 80.335,Z 363.528,A -85,B 0,C 180,E1 -28327.172,E2 -28327.172} C_VEL
LIN {X 0,Y 83.377,Z 368.335,A -85,B 0,C 180,E1 -28330.526,E2 -28330.526} C_VEL
LIN {X 0,Y 88.702,Z 378.378,A -85,B 0,C 180,E1 -28335.726,E2 -28335.726} C_VEL
LIN {X 0,Y 93.769,Z 391.651,A -85,B 0,C 180,E1 -28340.325,E2 -28340.325} C_VEL
LIN {X 0,Y 95.008,Z 395.252,A -85,B 0,C 180,E1 -28341.401,E2 -28341.401} C_VEL
LIN {X 0,Y 90.507,Z 433.466,A -85,B 0,C 180,E1 -28344.216,E2 -28344.216} C_VEL
LIN {X 0,Y 88.068,Z 447.158,A -85,B 0,C 180,E1 -28345.999,E2 -28345.999} C_VEL
LIN {X 0,Y 84.735,Z 460.38,A -85,B 0,C 180,E1 -28348.564,E2 -28348.564} C_VEL
LIN {X 0,Y 80.961,Z 472.296,A -85,B 0,C 180,E1 -28351.868,E2 -28351.868} C_VEL
LIN {X 0,Y 76.69,Z 484.057,A -85,B 0,C 180,E1 -28356.448,E2 -28356.448} C_VEL
LIN {X 0,Y 72.023,Z 495.36,A -85,B 0,C 180,E1 -28362.624,E2 -28362.624} C_VEL
LIN {X 0,Y 68.36,Z 504.235,A -85,B 0,C 180,E1 -28369.27,E2 -28369.27} C_VEL
LIN {X 0,Y 65.327,Z 512.338,A -85,B 0,C 180,E1 -28377.378,E2 -28377.378} C_VEL
LIN {X 0,Y 63.244,Z 518.869,A -85,B 0,C 180,E1 -28385.967,E2 -28385.967} C_VEL
LIN {X 0,Y 62.234,Z 525.416,A -85,B 0,C 180,E1 -28397.344,E2 -28397.344} C_VEL
LIN {X 0,Y 63.398,Z 530.525,A -85,B 0,C 180,E1 -28409.035,E2 -28409.035} C_VEL
LIN {X 0,Y 67.082,Z 534.314,A -85,B 0,C 180,E1 -28420.555,E2 -28420.555} C_VEL
LIN {X 0,Y 71.676,Z 536.327,A -85,B 0,C 180,E1 -28428.689,E2 -28428.689} C_VEL
LIN {X 0,Y 77.523,Z 537.459,A -85,B 0,C 180,E1 -28435.764,E2 -28435.764} C_VEL
LIN {X 0,Y 84.378,Z 537.718,A -85,B 0,C 180,E1 -28441.726,E2 -28441.726} C_VEL
LIN {X 0,Y 95.313,Z 536.69,A -85,B 0,C 180,E1 -28448.479,E2 -28448.479} C_VEL
LIN {X 0,Y 102.552,Z 535.227,A -85,B 0,C 180,E1 -28451.863,E2 -28451.863} C_VEL
LIN {X 0,Y 114.082,Z 531.785,A -85,B 0,C 180,E1 -28456.095,E2 -28456.095} C_VEL
LIN {X 0,Y 122.223,Z 528.548,A -85,B 0,C 180,E1 -28458.436,E2 -28458.436} C_VEL
LIN {X 0,Y 132.799,Z 523.279,A -85,B 0,C 180,E1 -28460.972,E2 -28460.972} C_VEL
LIN {X 0,Y 139.803,Z 519.038,A -85,B 0,C 180,E1 -28462.381,E2 -28462.381} C_VEL
LIN {X 0,Y 137.638,Z 520.521,A -85,B 0,C 180,E1 -28463.2,E2 -28463.2} C_VEL
LIN {X 0,Y 128.028,Z 526.179,A -85,B 0,C 180,E1 -28465.072,E2 -28465.072} C_VEL
LIN {X 0,Y 118.606,Z 530.737,A -85,B 0,C 180,E1 -28467.271,E2 -28467.271} C_VEL
LIN {X 0,Y 106.652,Z 535.293,A -85,B 0,C 180,E1 -28471.054,E2 -28471.054} C_VEL
LIN {X 0,Y 95.322,Z 538.347,A -85,B 0,C 180,E1 -28475.801,E2 -28475.801} C_VEL
LIN {X 0,Y 85.06,Z 539.997,A -85,B 0,C 180,E1 -28481.956,E2 -28481.956} C_VEL
LIN {X 0,Y 76.153,Z 540.262,A -85,B 0,C 180,E1 -28489.755,E2 -28489.755} C_VEL
LIN {X 0,Y 69.092,Z 539.126,A -85,B 0,C 180,E1 -28499.426,E2 -28499.426} C_VEL
LIN {X 0,Y 64.822,Z 536.653,A -85,B 0,C 180,E1 -28511.015,E2 -28511.015} C_VEL
LIN {X 0,Y 63.441,Z 533.764,A -85,B 0,C 180,E1 -28520.431,E2 -28520.431} C_VEL
LIN {X 0,Y 63.424,Z 531.766,A -85,B 0,C 180,E1 -28525.761,E2 -28525.761} C_VEL
LIN {X 0,Y 63.44,Z 529.886,A -85,B 0,C 180,E1 -28529.996,E2 -28529.996} C_VEL
LIN {X 0,Y 63.54,Z 524.595,A -85,B 0,C 180,E1 -28539.546,E2 -28539.546} C_VEL
LIN {X 0,Y 65.003,Z 517.879,A -85,B 0,C 180,E1 -28548.922,E2 -28548.922} C_VEL
LIN {X 0,Y 67.978,Z 509.48,A -85,B 0,C 180,E1 -28557.721,E2 -28557.721} C_VEL
LIN {X 0,Y 71.453,Z 500.799,A -85,B 0,C 180,E1 -28564.437,E2 -28564.437} C_VEL
LIN {X 0,Y 75.361,Z 491.303,A -85,B 0,C 180,E1 -28569.873,E2 -28569.873} C_VEL
LIN {X 0,Y 79.903,Z 479.624,A -85,B 0,C 180,E1 -28574.716,E2 -28574.716} C_VEL
LIN {X 0,Y 83.888,Z 467.626,A -85,B 0,C 180,E1 -28578.214,E2 -28578.214} C_VEL
LIN {X 0,Y 87.317,Z 455.136,A -85,B 0,C 180,E1 -28580.773,E2 -28580.773} C_VEL
LIN {X 0,Y 89.998,Z 441.796,A -85,B 0,C 180,E1 -28582.603,E2 -28582.603} C_VEL
LIN {X 0,Y 92.463,Z 421.829,A -85,B 0,C 180,E1 -28584.261,E2 -28584.261} C_VEL
LIN {X 0,Y 94.701,Z 400.821,A -85,B 0,C 180,E1 -28585.833,E2 -28585.833} C_VEL
LIN {X 0,Y 90.449,Z 385.13,A -85,B 0,C 180,E1 -28590.123,E2 -28590.123} C_VEL
LIN {X 0,Y 87.969,Z 378.444,A -85,B 0,C 180,E1 -28592.514,E2 -28592.514} C_VEL
LIN {X 0,Y 83.517,Z 369.446,A -85,B 0,C 180,E1 -28596.96,E2 -28596.96} C_VEL
LIN {X 0,Y 80.371,Z 363.902,A -85,B 0,C 180,E1 -28600.532,E2 -28600.532} C_VEL
LIN {X 0,Y 76.369,Z 357.282,A -85,B 0,C 180,E1 -28605.699,E2 -28605.699} C_VEL
LIN {X 0,Y 74.036,Z 353.821,A -85,B 0,C 180,E1 -28609.23,E2 -28609.23} C_VEL
LIN {X 0,Y 73.196,Z 352.481,A -85,B 0,C 180,E1 -28610.677,E2 -28610.677} C_VEL
LIN {X 0,Y 71.026,Z 349.57,A -85,B 0,C 180,E1 -28614.714,E2 -28614.714} C_VEL
LIN {X 0,Y 70.272,Z 347.827,A -85,B 0,C 180,E1 -28616.487,E2 -28616.487} C_VEL
LIN {X 0,Y 67.797,Z 345.868,A -85,B 0,C 180,E1 -28622.13,E2 -28622.13} C_VEL
LIN {X 0,Y 66.135,Z 345.274,A -85,B 0,C 180,E1 -28626.963,E2 -28626.963} C_VEL
LIN {X 0,Y 64.706,Z 345.801,A -85,B 0,C 180,E1 -28632.014,E2 -28632.014} C_VEL
LIN {X 0,Y 63.002,Z 348.826,A -85,B 0,C 180,E1 -28646.207,E2 -28646.207} C_VEL
LIN {X 0,Y 63.186,Z 349.129,A -85,B 0,C 180,E1 -28649.864,E2 -28649.864} C_VEL
LIN {X 0,Y 63.786,Z 349.439,A -85,B 0,C 180,E1 -28654.382,E2 -28654.382} C_VEL
LIN {X 0,Y 65.047,Z 352.542,A -85,B 0,C 180,E1 -28661.196,E2 -28661.196} C_VEL
LIN {X 0,Y 67.689,Z 355.013,A -85,B 0,C 180,E1 -28668.902,E2 -28668.902} C_VEL
LIN {X 0,Y 69.598,Z 358.256,A -85,B 0,C 180,E1 -28673.365,E2 -28673.365} C_VEL
LIN {X 0,Y 71.198,Z 359.868,A -85,B 0,C 180,E1 -28676.199,E2 -28676.199} C_VEL
LIN {X 0,Y 74.347,Z 365.001,A -85,B 0,C 180,E1 -28681.532,E2 -28681.532} C_VEL
LIN {X 0,Y 78.488,Z 371.447,A -85,B 0,C 180,E1 -28687.009,E2 -28687.009} C_VEL
LIN {X 0,Y 83.951,Z 382.042,A -85,B 0,C 180,E1 -28693.178,E2 -28693.178} C_VEL
LIN {X 0,Y 88.662,Z 394.954,A -85,B 0,C 180,E1 -28698.036,E2 -28698.036} C_VEL
LIN {X 0,Y 89.357,Z 397.141,A -85,B 0,C 180,E1 -28698.719,E2 -28698.719} C_VEL
LIN {X 0,Y 84.85,Z 433.325,A -85,B 0,C 180,E1 -28701.419,E2 -28701.419} C_VEL
LIN {X 0,Y 82.263,Z 447.15,A -85,B 0,C 180,E1 -28703.255,E2 -28703.255} C_VEL
LIN {X 0,Y 78.876,Z 459.975,A -85,B 0,C 180,E1 -28705.784,E2 -28705.784} C_VEL
LIN {X 0,Y 75.063,Z 471.483,A -85,B 0,C 180,E1 -28709.049,E2 -28709.049} C_VEL
LIN {X 0,Y 70.442,Z 483.502,A -85,B 0,C 180,E1 -28713.856,E2 -28713.856} C_VEL
LIN {X 0,Y 66.293,Z 493.082,A -85,B 0,C 180,E1 -28719.154,E2 -28719.154} C_VEL
LIN {X 0,Y 62.065,Z 502.623,A -85,B 0,C 180,E1 -28726.449,E2 -28726.449} C_VEL
LIN {X 0,Y 58.809,Z 510.581,A -85,B 0,C 180,E1 -28734.726,E2 -28734.726} C_VEL
LIN {X 0,Y 56.233,Z 518.088,A -85,B 0,C 180,E1 -28745.185,E2 -28745.185} C_VEL
LIN {X 0,Y 55.213,Z 523.666,A -85,B 0,C 180,E1 -28755.486,E2 -28755.486} C_VEL
LIN {X 0,Y 55.678,Z 527.971,A -85,B 0,C 180,E1 -28765.386,E2 -28765.386} C_VEL
LIN {X 0,Y 58.91,Z 532.78,A -85,B 0,C 180,E1 -28779.027,E2 -28779.027} C_VEL
LIN {X 0,Y 64.27,Z 535.735,A -85,B 0,C 180,E1 -28789.809,E2 -28789.809} C_VEL
LIN {X 0,Y 72.861,Z 537.639,A -85,B 0,C 180,E1 -28799.999,E2 -28799.999} C_VEL
LIN {X 0,Y 79.176,Z 538.048,A -85,B 0,C 180,E1 -28805.091,E2 -28805.091} C_VEL
LIN {X 0,Y 86.094,Z 537.82,A -85,B 0,C 180,E1 -28809.395,E2 -28809.395} C_VEL
LIN {X 0,Y 93.863,Z 536.92,A -85,B 0,C 180,E1 -28813.241,E2 -28813.241} C_VEL
LIN {X 0,Y 102.723,Z 535.176,A -85,B 0,C 180,E1 -28816.69,E2 -28816.69} C_VEL
LIN {X 0,Y 114.705,Z 531.575,A -85,B 0,C 180,E1 -28820.3,E2 -28820.3} C_VEL
LIN {X 0,Y 121.166,Z 529.072,A -85,B 0,C 180,E1 -28821.863,E2 -28821.863} C_VEL
LIN {X 0,Y 121.979,Z 528.793,A -85,B 0,C 180,E1 -28822.796,E2 -28822.796} C_VEL
LIN {X 0,Y 112.446,Z 532.735,A -85,B 0,C 180,E1 -28825.002,E2 -28825.002} C_VEL
LIN {X 0,Y 103.179,Z 535.741,A -85,B 0,C 180,E1 -28827.685,E2 -28827.685} C_VEL
LIN {X 0,Y 91.35,Z 538.496,A -85,B 0,C 180,E1 -28832.186,E2 -28832.186} C_VEL
LIN {X 0,Y 80.473,Z 539.828,A -85,B 0,C 180,E1 -28838.183,E2 -28838.183} C_VEL
LIN {X 0,Y 70.878,Z 539.817,A -85,B 0,C 180,E1 -28846.041,E2 -28846.041} C_VEL
LIN {X 0,Y 63.086,Z 538.461,A -85,B 0,C 180,E1 -28856.146,E2 -28856.146} C_VEL
LIN {X 0,Y 58.188,Z 535.699,A -85,B 0,C 180,E1 -28868.752,E2 -28868.752} C_VEL
LIN {X 0,Y 56.43,Z 531.416,A -85,B 0,C 180,E1 -28882.841,E2 -28882.841} C_VEL
LIN {X 0,Y 56.408,Z 528.565,A -85,B 0,C 180,E1 -28889.996,E2 -28889.996} C_VEL
LIN {X 0,Y 56.607,Z 523.006,A -85,B 0,C 180,E1 -28900.729,E2 -28900.729} C_VEL
LIN {X 0,Y 58.367,Z 515.927,A -85,B 0,C 180,E1 -28911.171,E2 -28911.171} C_VEL
LIN {X 0,Y 61.821,Z 507.1,A -85,B 0,C 180,E1 -28920.764,E2 -28920.764} C_VEL
LIN {X 0,Y 65.74,Z 498.008,A -85,B 0,C 180,E1 -28927.926,E2 -28927.926} C_VEL
LIN {X 0,Y 70.078,Z 487.988,A -85,B 0,C 180,E1 -28933.584,E2 -28933.584} C_VEL
LIN {X 0,Y 74.463,Z 477.03,A -85,B 0,C 180,E1 -28938.005,E2 -28938.005} C_VEL
LIN {X 0,Y 78.243,Z 466.166,A -85,B 0,C 180,E1 -28941.148,E2 -28941.148} C_VEL
LIN {X 0,Y 81.766,Z 453.757,A -85,B 0,C 180,E1 -28943.682,E2 -28943.682} C_VEL
LIN {X 0,Y 84.486,Z 440.45,A -85,B 0,C 180,E1 -28945.487,E2 -28945.487} C_VEL
LIN {X 0,Y 87.969,Z 412.831,A -85,B 0,C 180,E1 -28947.695,E2 -28947.695} C_VEL
LIN {X 0,Y 89.046,Z 402.225,A -85,B 0,C 180,E1 -28948.562,E2 -28948.562} C_VEL
LIN {X 0,Y 85.492,Z 388.538,A -85,B 0,C 180,E1 -28952.585,E2 -28952.585} C_VEL
LIN {X 0,Y 83.409,Z 382.56,A -85,B 0,C 180,E1 -28954.906,E2 -28954.906} C_VEL
LIN {X 0,Y 79.458,Z 374.028,A -85,B 0,C 180,E1 -28959.473,E2 -28959.473} C_VEL
LIN {X 0,Y 76.207,Z 368.139,A -85,B 0,C 180,E1 -28963.601,E2 -28963.601} C_VEL
LIN {X 0,Y 73.046,Z 362.725,A -85,B 0,C 180,E1 -28968.337,E2 -28968.337} C_VEL
LIN {X 0,Y 70.586,Z 358.557,A -85,B 0,C 180,E1 -28972.852,E2 -28972.852} C_VEL
LIN {X 0,Y 68.391,Z 355.225,A -85,B 0,C 180,E1 -28977.482,E2 -28977.482} C_VEL
LIN {X 0,Y 67.835,Z 354.165,A -85,B 0,C 180,E1 -28978.913,E2 -28978.913} C_VEL
LIN {X 0,Y 64.585,Z 350.358,A -85,B 0,C 180,E1 -28989.399,E2 -28989.399} C_VEL
LIN {X 0,Y 64.185,Z 349.174,A -85,B 0,C 180,E1 -28991.77,E2 -28991.77} C_VEL
LIN {X 0,Y 63.186,Z 349.129,A -85,B 0,C 180,E1 -29009.864,E2 -29009.864} C_VEL
LIN {X 0,Y 63.417,Z 349.937,A -85,B 0,C 180,E1 -29012.695,E2 -29012.695} C_VEL
LIN {X 0,Y 63.629,Z 352.641,A -85,B 0,C 180,E1 -29016.127,E2 -29016.127} C_VEL
LIN {X 0,Y 64.292,Z 359.323,A -85,B 0,C 180,E1 -29022.4,E2 -29022.4} C_VEL
LIN {X 0,Y 65.145,Z 361.067,A -85,B 0,C 180,E1 -29025.568,E2 -29025.568} C_VEL
LIN {X 0,Y 65.669,Z 361.696,A -85,B 0,C 180,E1 -29027.078,E2 -29027.078} C_VEL
LIN {X 0,Y 67.826,Z 365.151,A -85,B 0,C 180,E1 -29032.51,E2 -29032.51} C_VEL
LIN {X 0,Y 68.903,Z 366.641,A -85,B 0,C 180,E1 -29034.688,E2 -29034.688} C_VEL
LIN {X 0,Y 71.31,Z 370.663,A -85,B 0,C 180,E1 -29039.157,E2 -29039.157} C_VEL
LIN {X 0,Y 75.356,Z 377.535,A -85,B 0,C 180,E1 -29045.259,E2 -29045.259} C_VEL
LIN {X 0,Y 79.834,Z 387.075,A -85,B 0,C 180,E1 -29050.933,E2 -29050.933} C_VEL
LIN {X 0,Y 83.793,Z 398.727,A -85,B 0,C 180,E1 -29055.659,E2 -29055.659} C_VEL
LIN {X 0,Y 79.42,Z 432.876,A -85,B 0,C 180,E1 -29058.248,E2 -29058.248} C_VEL
LIN {X 0,Y 77.12,Z 445.169,A -85,B 0,C 180,E1 -29059.833,E2 -29059.833} C_VEL
LIN {X 0,Y 73.409,Z 458.874,A -85,B 0,C 180,E1 -29062.439,E2 -29062.439} C_VEL
LIN {X 0,Y 69.459,Z 470.415,A -85,B 0,C 180,E1 -29065.665,E2 -29065.665} C_VEL
LIN {X 0,Y 64.638,Z 482.335,A -85,B 0,C 180,E1 -29070.493,E2 -29070.493} C_VEL
LIN {X 0,Y 59.618,Z 493.231,A -85,B 0,C 180,E1 -29076.774,E2 -29076.774} C_VEL
LIN {X 0,Y 55.075,Z 502.783,A -85,B 0,C 180,E1 -29084.791,E2 -29084.791} C_VEL
LIN {X 0,Y 51.627,Z 510.728,A -85,B 0,C 180,E1 -29094.109,E2 -29094.109} C_VEL
LIN {X 0,Y 49.146,Z 517.559,A -85,B 0,C 180,E1 -29104.896,E2 -29104.896} C_VEL
LIN {X 0,Y 48.149,Z 523.354,A -85,B 0,C 180,E1 -29116.878,E2 -29116.878} C_VEL
LIN {X 0,Y 49.633,Z 529.234,A -85,B 0,C 180,E1 -29132.279,E2 -29132.279} C_VEL
LIN {X 0,Y 53.574,Z 533.146,A -85,B 0,C 180,E1 -29144.788,E2 -29144.788} C_VEL
LIN {X 0,Y 58.095,Z 535.36,A -85,B 0,C 180,E1 -29153.05,E2 -29153.05} C_VEL
LIN {X 0,Y 63.563,Z 536.976,A -85,B 0,C 180,E1 -29159.998,E2 -29159.998} C_VEL
LIN {X 0,Y 70.725,Z 538.052,A -85,B 0,C 180,E1 -29166.407,E2 -29166.407} C_VEL
LIN {X 0,Y 78.961,Z 538.35,A -85,B 0,C 180,E1 -29171.73,E2 -29171.73} C_VEL
LIN {X 0,Y 87.735,Z 537.85,A -85,B 0,C 180,E1 -29175.992,E2 -29175.992} C_VEL
LIN {X 0,Y 100.344,Z 535.852,A -85,B 0,C 180,E1 -29180.498,E2 -29180.498} C_VEL
LIN {X 0,Y 106.243,Z 534.43,A -85,B 0,C 180,E1 -29182.16,E2 -29182.16} C_VEL
LIN {X 0,Y 106.438,Z 534.394,A -85,B 0,C 180,E1 -29182.416,E2 -29182.416} C_VEL
LIN {X 0,Y 93.856,Z 537.52,A -85,B 0,C 180,E1 -29186.024,E2 -29186.024} C_VEL
LIN {X 0,Y 81.904,Z 539.255,A -85,B 0,C 180,E1 -29190.894,E2 -29190.894} C_VEL
LIN {X 0,Y 70.939,Z 539.661,A -85,B 0,C 180,E1 -29197.569,E2 -29197.569} C_VEL
LIN {X 0,Y 61.394,Z 538.691,A -85,B 0,C 180,E1 -29206.614,E2 -29206.614} C_VEL
LIN {X 0,Y 57.341,Z 537.689,A -85,B 0,C 180,E1 -29212.201,E2 -29212.201} C_VEL
LIN {X 0,Y 51.676,Z 534.682,A -85,B 0,C 180,E1 -29225.916,E2 -29225.916} C_VEL
LIN {X 0,Y 49.508,Z 530.137,A -85,B 0,C 180,E1 -29241.834,E2 -29241.834} C_VEL
LIN {X 0,Y 49.395,Z 527.092,A -85,B 0,C 180,E1 -29249.995,E2 -29249.995} C_VEL
LIN {X 0,Y 49.706,Z 521.264,A -85,B 0,C 180,E1 -29262.24,E2 -29262.24} C_VEL
LIN {X 0,Y 51.849,Z 513.893,A -85,B 0,C 180,E1 -29273.989,E2 -29273.989} C_VEL
LIN {X 0,Y 55.09,Z 506.335,A -85,B 0,C 180,E1 -29282.827,E2 -29282.827} C_VEL
LIN {X 0,Y 59.87,Z 496.087,A -85,B 0,C 180,E1 -29291.318,E2 -29291.318} C_VEL
LIN {X 0,Y 65.184,Z 484.456,A -85,B 0,C 180,E1 -29297.832,E2 -29297.832} C_VEL
LIN {X 0,Y 69.953,Z 472.616,A -85,B 0,C 180,E1 -29302.29,E2 -29302.29} C_VEL
LIN {X 0,Y 74.365,Z 459.496,A -85,B 0,C 180,E1 -29305.637,E2 -29305.637} C_VEL
LIN {X 0,Y 77.81,Z 446.014,A -85,B 0,C 180,E1 -29307.856,E2 -29307.856} C_VEL
LIN {X 0,Y 79.993,Z 433.175,A -85,B 0,C 180,E1 -29309.238,E2 -29309.238} C_VEL
LIN {X 0,Y 83.559,Z 403.812,A -85,B 0,C 180,E1 -29311.512,E2 -29311.512} C_VEL
LIN {X 0,Y 80.523,Z 391.215,A -85,B 0,C 180,E1 -29315.602,E2 -29315.602} C_VEL
LIN {X 0,Y 78.696,Z 385.835,A -85,B 0,C 180,E1 -29317.983,E2 -29317.983} C_VEL
LIN {X 0,Y 75.051,Z 377.646,A -85,B 0,C 180,E1 -29322.825,E2 -29322.825} C_VEL
LIN {X 0,Y 70.537,Z 369.027,A -85,B 0,C 180,E1 -29330.068,E2 -29330.068} C_VEL
LIN {X 0,Y 67.879,Z 364.432,A -85,B 0,C 180,E1 -29335.449,E2 -29335.449} C_VEL
LIN {X 0,Y 65.544,Z 360.345,A -85,B 0,C 180,E1 -29341.538,E2 -29341.538} C_VEL
LIN {X 0,Y 63.065,Z 357.132,A -85,B 0,C 180,E1 -29350.909,E2 -29350.909} C_VEL
LIN {X 0,Y 62.774,Z 356.187,A -85,B 0,C 180,E1 -29352.941,E2 -29352.941} C_VEL
LIN {X 0,Y 62.258,Z 356.188,A -85,B 0,C 180,E1 -29371.791,E2 -29371.791} C_VEL
LIN {X 0,Y 62.449,Z 356.702,A -85,B 0,C 180,E1 -29373.597,E2 -29373.597} C_VEL
LIN {X 0,Y 63.908,Z 359.912,A -85,B 0,C 180,E1 -29381.528,E2 -29381.528} C_VEL
LIN {X 0,Y 65.145,Z 361.067,A -85,B 0,C 180,E1 -29385.568,E2 -29385.568} C_VEL
LIN {X 0,Y 66.232,Z 362.451,A -85,B 0,C 180,E1 -29388.59,E2 -29388.59} C_VEL
LIN {X 0,Y 67.677,Z 365.909,A -85,B 0,C 180,E1 -29392.469,E2 -29392.469} C_VEL
LIN {X 0,Y 68.876,Z 370.325,A -85,B 0,C 180,E1 -29395.674,E2 -29395.674} C_VEL
LIN {X 0,Y 72.251,Z 383.717,A -85,B 0,C 180,E1 -29403.331,E2 -29403.331} C_VEL
LIN {X 0,Y 75.57,Z 391.401,A -85,B 0,C 180,E1 -29408.165,E2 -29408.165} C_VEL
LIN {X 0,Y 78.561,Z 400.57,A -85,B 0,C 180,E1 -29412.271,E2 -29412.271} C_VEL
LIN {X 0,Y 74.117,Z 433.309,A -85,B 0,C 180,E1 -29414.713,E2 -29414.713} C_VEL
LIN {X 0,Y 71.202,Z 447.372,A -85,B 0,C 180,E1 -29416.578,E2 -29416.578} C_VEL
LIN {X 0,Y 67.48,Z 460.043,A -85,B 0,C 180,E1 -29419.123,E2 -29419.123} C_VEL
LIN {X 0,Y 63.226,Z 471.464,A -85,B 0,C 180,E1 -29422.502,E2 -29422.502} C_VEL
LIN {X 0,Y 58.237,Z 482.873,A -85,B 0,C 180,E1 -29427.41,E2 -29427.41} C_VEL
LIN {X 0,Y 53.128,Z 493.167,A -85,B 0,C 180,E1 -29433.797,E2 -29433.797} C_VEL
LIN {X 0,Y 48.002,Z 503.122,A -85,B 0,C 180,E1 -29443.015,E2 -29443.015} C_VEL
LIN {X 0,Y 44.074,Z 511.638,A -85,B 0,C 180,E1 -29454.613,E2 -29454.613} C_VEL
LIN {X 0,Y 41.516,Z 518.949,A -85,B 0,C 180,E1 -29468.65,E2 -29468.65} C_VEL
LIN {X 0,Y 41.296,Z 524.471,A -85,B 0,C 180,E1 -29482.657,E2 -29482.657} C_VEL
LIN {X 0,Y 44.551,Z 530.414,A -85,B 0,C 180,E1 -29501.192,E2 -29501.192} C_VEL
LIN {X 0,Y 49.575,Z 533.798,A -85,B 0,C 180,E1 -29512.943,E2 -29512.943} C_VEL
LIN {X 0,Y 56.273,Z 536.284,A -85,B 0,C 180,E1 -29522.309,E2 -29522.309} C_VEL
LIN {X 0,Y 64.129,Z 537.867,A -85,B 0,C 180,E1 -29529.466,E2 -29529.466} C_VEL
LIN {X 0,Y 75.298,Z 538.679,A -85,B 0,C 180,E1 -29536.259,E2 -29536.259} C_VEL
LIN {X 0,Y 87.016,Z 538.16,A -85,B 0,C 180,E1 -29541.068,E2 -29541.068} C_VEL
LIN {X 0,Y 88.856,Z 537.973,A -85,B 0,C 180,E1 -29541.681,E2 -29541.681} C_VEL
LIN {X 0,Y 86.388,Z 538.374,A -85,B 0,C 180,E1 -29543.446,E2 -29543.446} C_VEL
LIN {X 0,Y 76.222,Z 539.246,A -85,B 0,C 180,E1 -29547.452,E2 -29547.452} C_VEL
LIN {X 0,Y 66.848,Z 539.226,A -85,B 0,C 180,E1 -29552.741,E2 -29552.741} C_VEL
LIN {X 0,Y 56.454,Z 537.999,A -85,B 0,C 180,E1 -29561.668,E2 -29561.668} C_VEL
LIN {X 0,Y 48.232,Z 535.431,A -85,B 0,C 180,E1 -29574.343,E2 -29574.343} C_VEL
LIN {X 0,Y 43.432,Z 531.394,A -85,B 0,C 180,E1 -29591.112,E2 -29591.112} C_VEL
LIN {X 0,Y 42.541,Z 527.426,A -85,B 0,C 180,E1 -29604.781,E2 -29604.781} C_VEL
LIN {X 0,Y 42.344,Z 523.469,A -85,B 0,C 180,E1 -29615.242,E2 -29615.242} C_VEL
LIN {X 0,Y 43.505,Z 517.02,A -85,B 0,C 180,E1 -29628.844,E2 -29628.844} C_VEL
LIN {X 0,Y 46.884,Z 508.687,A -85,B 0,C 180,E1 -29641.639,E2 -29641.639} C_VEL
LIN {X 0,Y 51.134,Z 500.093,A -85,B 0,C 180,E1 -29650.751,E2 -29650.751} C_VEL
LIN {X 0,Y 55.896,Z 490.739,A -85,B 0,C 180,E1 -29657.613,E2 -29657.613} C_VEL
LIN {X 0,Y 61.324,Z 479.24,A -85,B 0,C 180,E1 -29663.336,E2 -29663.336} C_VEL
LIN {X 0,Y 65.926,Z 467.868,A -85,B 0,C 180,E1 -29667.081,E2 -29667.081} C_VEL
LIN {X 0,Y 70.314,Z 454.279,A -85,B 0,C 180,E1 -29670.102,E2 -29670.102} C_VEL
LIN {X 0,Y 73.39,Z 441.236,A -85,B 0,C 180,E1 -29671.947,E2 -29671.947} C_VEL
LIN {X 0,Y 75.962,Z 423.467,A -85,B 0,C 180,E1 -29673.518,E2 -29673.518} C_VEL
LIN {X 0,Y 78.252,Z 405.085,A -85,B 0,C 180,E1 -29674.962,E2 -29674.962} C_VEL
LIN {X 0,Y 75.623,Z 393.373,A -85,B 0,C 180,E1 -29679.239,E2 -29679.239} C_VEL
LIN {X 0,Y 73.491,Z 387.615,A -85,B 0,C 180,E1 -29682.342,E2 -29682.342} C_VEL
LIN {X 0,Y 70.556,Z 380.718,A -85,B 0,C 180,E1 -29687.115,E2 -29687.115} C_VEL
LIN {X 0,Y 67.327,Z 374.152,A -85,B 0,C 180,E1 -29693.44,E2 -29693.44} C_VEL
LIN {X 0,Y 65.365,Z 370.347,A -85,B 0,C 180,E1 -29698.119,E2 -29698.119} C_VEL
LIN {X 0,Y 63.587,Z 366.769,A -85,B 0,C 180,E1 -29703.702,E2 -29703.702} C_VEL
LIN {X 0,Y 61.545,Z 363.747,A -85,B 0,C 180,E1 -29712.823,E2 -29712.823} C_VEL
LIN {X 0,Y 61.342,Z 363.148,A -85,B 0,C 180,E1 -29714.489,E2 -29714.489} C_VEL
LIN {X 0,Y 61.037,Z 363.182,A -85,B 0,C 180,E1 -29731.21,E2 -29731.21} C_VEL
LIN {X 0,Y 62.333,Z 366.674,A -85,B 0,C 180,E1 -29740.181,E2 -29740.181} C_VEL
LIN {X 0,Y 63.703,Z 368.244,A -85,B 0,C 180,E1 -29745.039,E2 -29745.039} C_VEL
LIN {X 0,Y 66.383,Z 372.714,A -85,B 0,C 180,E1 -29752.384,E2 -29752.384} C_VEL
LIN {X 0,Y 68.979,Z 377.372,A -85,B 0,C 180,E1 -29757.704,E2 -29757.704} C_VEL
LIN {X 0,Y 72.081,Z 383.298,A -85,B 0,C 180,E1 -29763.051,E2 -29763.051} C_VEL
LIN {X 0,Y 72.251,Z 383.717,A -85,B 0,C 180,E1 -29763.331,E2 -29763.331} C_VEL
LIN {X 0,Y 73.426,Z 388.162,A -85,B 0,C 180,E1 -29765.509,E2 -29765.509} C_VEL
LIN {X 0,Y 73.933,Z 393.172,A -85,B 0,C 180,E1 -29767.015,E2 -29767.015} C_VEL
LIN {X 0,Y 73.663,Z 401.205,A -85,B 0,C 180,E1 -29768.342,E2 -29768.342} C_VEL
LIN {X 0,Y 73.347,Z 403.915,A -85,B 0,C 180,E1 -29768.583,E2 -29768.583} C_VEL
LIN {X 0,Y 68.9,Z 434.312,A -85,B 0,C 180,E1 -29770.782,E2 -29770.782} C_VEL
LIN {X 0,Y 65.869,Z 447.949,A -85,B 0,C 180,E1 -29772.596,E2 -29772.596} C_VEL
LIN {X 0,Y 61.918,Z 460.576,A -85,B 0,C 180,E1 -29775.125,E2 -29775.125} C_VEL
LIN {X 0,Y 56.802,Z 473.248,A -85,B 0,C 180,E1 -29778.999,E2 -29778.999} C_VEL
LIN {X 0,Y 51.73,Z 483.947,A -85,B 0,C 180,E1 -29783.93,E2 -29783.93} C_VEL
LIN {X 0,Y 46.043,Z 494.418,A -85,B 0,C 180,E1 -29791.098,E2 -29791.098} C_VEL
LIN {X 0,Y 40.744,Z 503.896,A -85,B 0,C 180,E1 -29801.195,E2 -29801.195} C_VEL
LIN {X 0,Y 37.221,Z 510.905,A -85,B 0,C 180,E1 -29812.194,E2 -29812.194} C_VEL
LIN {X 0,Y 34.53,Z 517.854,A -85,B 0,C 180,E1 -29827.641,E2 -29827.641} C_VEL
LIN {X 0,Y 34.396,Z 523.693,A -85,B 0,C 180,E1 -29844.828,E2 -29844.828} C_VEL
LIN {X 0,Y 37.058,Z 528.56,A -85,B 0,C 180,E1 -29861.504,E2 -29861.504} C_VEL
LIN {X 0,Y 42.312,Z 532.459,A -85,B 0,C 180,E1 -29875.327,E2 -29875.327} C_VEL
LIN {X 0,Y 51.454,Z 535.973,A -85,B 0,C 180,E1 -29887.849,E2 -29887.849} C_VEL
LIN {X 0,Y 58.657,Z 537.592,A -85,B 0,C 180,E1 -29893.863,E2 -29893.863} C_VEL
LIN {X 0,Y 70.608,Z 538.863,A -85,B 0,C 180,E1 -29900.546,E2 -29900.546} C_VEL
LIN {X 0,Y 72.568,Z 538.949,A -85,B 0,C 180,E1 -29901.372,E2 -29901.372} C_VEL
LIN {X 0,Y 72.388,Z 539.021,A -85,B 0,C 180,E1 -29902.851,E2 -29902.851} C_VEL
LIN {X 0,Y 63.292,Z 538.767,A -85,B 0,C 180,E1 -29907.328,E2 -29907.328} C_VEL
LIN {X 0,Y 52.016,Z 537.251,A -85,B 0,C 180,E1 -29915.831,E2 -29915.831} C_VEL
LIN {X 0,Y 42.703,Z 534.375,A -85,B 0,C 180,E1 -29928.822,E2 -29928.822} C_VEL
LIN {X 0,Y 36.89,Z 530.07,A -85,B 0,C 180,E1 -29947.596,E2 -29947.596} C_VEL
LIN {X 0,Y 35.634,Z 525.892,A -85,B 0,C 180,E1 -29963.766,E2 -29963.766} C_VEL
LIN {X 0,Y 35.391,Z 521.549,A -85,B 0,C 180,E1 -29976.842,E2 -29976.842} C_VEL
LIN {X 0,Y 36.911,Z 514.945,A -85,B 0,C 180,E1 -29992.377,E2 -29992.377} C_VEL
LIN {X 0,Y 41.072,Z 506.169,A -85,B 0,C 180,E1 -30006.783,E2 -30006.783} C_VEL
LIN {X 0,Y 46.04,Z 497.137,A -85,B 0,C 180,E1 -30016.469,E2 -30016.469} C_VEL
LIN {X 0,Y 51.41,Z 487.17,A -85,B 0,C 180,E1 -30023.422,E2 -30023.422} C_VEL
LIN {X 0,Y 56.735,Z 476.307,A -85,B 0,C 180,E1 -30028.382,E2 -30028.382} C_VEL
LIN {X 0,Y 61.654,Z 464.318,A -85,B 0,C 180,E1 -30032.05,E2 -30032.05} C_VEL
LIN {X 0,Y 65.666,Z 451.997,A -85,B 0,C 180,E1 -30034.49,E2 -30034.49} C_VEL
LIN {X 0,Y 68.891,Z 438.144,A -85,B 0,C 180,E1 -30036.269,E2 -30036.269} C_VEL
LIN {X 0,Y 73.303,Z 406.747,A -85,B 0,C 180,E1 -30038.726,E2 -30038.726} C_VEL
LIN {X 0,Y 71.127,Z 396.29,A -85,B 0,C 180,E1 -30042.935,E2 -30042.935} C_VEL
LIN {X 0,Y 68.213,Z 388.12,A -85,B 0,C 180,E1 -30048.295,E2 -30048.295} C_VEL
LIN {X 0,Y 64.892,Z 380.309,A -85,B 0,C 180,E1 -30055.636,E2 -30055.636} C_VEL
LIN {X 0,Y 62.943,Z 376.198,A -85,B 0,C 180,E1 -30061.171,E2 -30061.171} C_VEL
LIN {X 0,Y 61.677,Z 373.221,A -85,B 0,C 180,E1 -30066.148,E2 -30066.148} C_VEL
LIN {X 0,Y 60.032,Z 370.14,A -85,B 0,C 180,E1 -30075.522,E2 -30075.522} C_VEL
LIN {X 0,Y 59.757,Z 370.192,A -85,B 0,C 180,E1 -30089.991,E2 -30089.991} C_VEL
LIN {X 0,Y 61.042,Z 373.759,A -85,B 0,C 180,E1 -30099.856,E2 -30099.856} C_VEL
LIN {X 0,Y 61.898,Z 374.888,A -85,B 0,C 180,E1 -30103.157,E2 -30103.157} C_VEL
LIN {X 0,Y 64.126,Z 379.136,A -85,B 0,C 180,E1 -30110.327,E2 -30110.327} C_VEL
LIN {X 0,Y 66.783,Z 384.386,A -85,B 0,C 180,E1 -30116.47,E2 -30116.47} C_VEL
LIN {X 0,Y 68.946,Z 389.094,A -85,B 0,C 180,E1 -30120.673,E2 -30120.673} C_VEL
LIN {X 0,Y 71.557,Z 395.957,A -85,B 0,C 180,E1 -30125.24,E2 -30125.24} C_VEL
LIN {X 0,Y 73.499,Z 402.425,A -85,B 0,C 180,E1 -30128.431,E2 -30128.431} C_VEL
LIN {X 0,Y 73.347,Z 403.915,A -85,B 0,C 180,E1 -30128.583,E2 -30128.583} C_VEL
LIN {X 0,Y 72.147,Z 409.7,A -85,B 0,C 180,E1 -30128.601,E2 -30128.601} C_VEL
LIN {X 0,Y 65.784,Z 428.294,A -85,B 0,C 180,E1 -30126.199,E2 -30126.199} C_VEL
LIN {X 0,Y 64.314,Z 434.039,A -85,B 0,C 180,E1 -30126.14,E2 -30126.14} C_VEL
LIN {X 0,Y 61.148,Z 447.675,A -85,B 0,C 180,E1 -30127.815,E2 -30127.815} C_VEL
LIN {X 0,Y 57.02,Z 460.328,A -85,B 0,C 180,E1 -30130.191,E2 -30130.191} C_VEL
LIN {X 0,Y 52.267,Z 471.648,A -85,B 0,C 180,E1 -30133.402,E2 -30133.402} C_VEL
LIN {X 0,Y 47.091,Z 482.018,A -85,B 0,C 180,E1 -30137.836,E2 -30137.836} C_VEL
LIN {X 0,Y 40.98,Z 492.545,A -85,B 0,C 180,E1 -30144.755,E2 -30144.755} C_VEL
LIN {X 0,Y 34.785,Z 502.539,A -85,B 0,C 180,E1 -30155.556,E2 -30155.556} C_VEL
LIN {X 0,Y 30.047,Z 510.903,A -85,B 0,C 180,E1 -30170.662,E2 -30170.662} C_VEL
LIN {X 0,Y 27.344,Z 517.747,A -85,B 0,C 180,E1 -30189.543,E2 -30189.543} C_VEL
LIN {X 0,Y 27.676,Z 523.253,A -85,B 0,C 180,E1 -30209.473,E2 -30209.473} C_VEL
LIN {X 0,Y 30.734,Z 527.658,A -85,B 0,C 180,E1 -30226.778,E2 -30226.778} C_VEL
LIN {X 0,Y 38.956,Z 532.706,A -85,B 0,C 180,E1 -30245.173,E2 -30245.173} C_VEL
LIN {X 0,Y 49.66,Z 536.253,A -85,B 0,C 180,E1 -30256.44,E2 -30256.44} C_VEL
LIN {X 0,Y 57.627,Z 537.888,A -85,B 0,C 180,E1 -30261.46,E2 -30261.46} C_VEL
LIN {X 0,Y 54.177,Z 537.47,A -85,B 0,C 180,E1 -30264.753,E2 -30264.753} C_VEL
LIN {X 0,Y 42.64,Z 535.005,A -85,B 0,C 180,E1 -30274.492,E2 -30274.492} C_VEL
LIN {X 0,Y 33.588,Z 531.19,A -85,B 0,C 180,E1 -30291.109,E2 -30291.109} C_VEL
LIN {X 0,Y 29.062,Z 525.741,A -85,B 0,C 180,E1 -30315.997,E2 -30315.997} C_VEL
LIN {X 0,Y 28.456,Z 522.191,A -85,B 0,C 180,E1 -30329.992,E2 -30329.992} C_VEL
LIN {X 0,Y 29.472,Z 515.394,A -85,B 0,C 180,E1 -30350.95,E2 -30350.95} C_VEL
LIN {X 0,Y 33.712,Z 506.832,A -85,B 0,C 180,E1 -30368.703,E2 -30368.703} C_VEL
LIN {X 0,Y 39.057,Z 498.033,A -85,B 0,C 180,E1 -30379.876,E2 -30379.876} C_VEL
LIN {X 0,Y 44.811,Z 488.384,A -85,B 0,C 180,E1 -30387.448,E2 -30387.448} C_VEL
LIN {X 0,Y 50.447,Z 477.868,A -85,B 0,C 180,E1 -30392.628,E2 -30392.628} C_VEL
LIN {X 0,Y 55.657,Z 466.349,A -85,B 0,C 180,E1 -30396.264,E2 -30396.264} C_VEL
LIN {X 0,Y 60.254,Z 453.519,A -85,B 0,C 180,E1 -30398.914,E2 -30398.914} C_VEL
LIN {X 0,Y 63.541,Z 441.031,A -85,B 0,C 180,E1 -30400.518,E2 -30400.518} C_VEL
LIN {X 0,Y 66.495,Z 422.776,A -85,B 0,C 180,E1 -30402.02,E2 -30402.02} C_VEL
LIN {X 0,Y 68.568,Z 408.242,A -85,B 0,C 180,E1 -30403.045,E2 -30403.045} C_VEL
LIN {X 0,Y 66.961,Z 399.344,A -85,B 0,C 180,E1 -30407.081,E2 -30407.081} C_VEL
LIN {X 0,Y 64.641,Z 392.269,A -85,B 0,C 180,E1 -30412.374,E2 -30412.374} C_VEL
LIN {X 0,Y 62.219,Z 385.829,A -85,B 0,C 180,E1 -30418.965,E2 -30418.965} C_VEL
LIN {X 0,Y 60.697,Z 381.928,A -85,B 0,C 180,E1 -30424.571,E2 -30424.571} C_VEL
LIN {X 0,Y 60.007,Z 379.829,A -85,B 0,C 180,E1 -30428.067,E2 -30428.067} C_VEL
LIN {X 0,Y 58.722,Z 377.124,A -85,B 0,C 180,E1 -30436.788,E2 -30436.788} C_VEL
LIN {X 0,Y 58.504,Z 377.357,A -85,B 0,C 180,E1 -30449.048,E2 -30449.048} C_VEL
LIN {X 0,Y 60.102,Z 381.484,A -85,B 0,C 180,E1 -30461.085,E2 -30461.085} C_VEL
LIN {X 0,Y 61.903,Z 385.337,A -85,B 0,C 180,E1 -30467.91,E2 -30467.91} C_VEL
LIN {X 0,Y 64.759,Z 391.893,A -85,B 0,C 180,E1 -30475.537,E2 -30475.537} C_VEL
LIN {X 0,Y 67.517,Z 399.523,A -85,B 0,C 180,E1 -30481.445,E2 -30481.445} C_VEL
LIN {X 0,Y 68.795,Z 404.549,A -85,B 0,C 180,E1 -30484.16,E2 -30484.16} C_VEL
LIN {X 0,Y 64.314,Z 434.039,A -85,B 0,C 180,E1 -30486.14,E2 -30486.14} C_VEL
LIN {X 0,Y 62.694,Z 439.732,A -85,B 0,C 180,E1 -30486.17,E2 -30486.17} C_VEL
LIN {X 0,Y 58.599,Z 448.72,A -85,B 0,C 180,E1 -30485.212,E2 -30485.212} C_VEL
LIN {X 0,Y 53.938,Z 457.479,A -85,B 0,C 180,E1 -30484.472,E2 -30484.472} C_VEL
LIN {X 0,Y 51.408,Z 462.819,A -85,B 0,C 180,E1 -30485.06,E2 -30485.06} C_VEL
LIN {X 0,Y 45.749,Z 474.907,A -85,B 0,C 180,E1 -30488.569,E2 -30488.569} C_VEL
LIN {X 0,Y 39.829,Z 485.333,A -85,B 0,C 180,E1 -30493.344,E2 -30493.344} C_VEL
LIN {X 0,Y 32.453,Z 496.537,A -85,B 0,C 180,E1 -30502.229,E2 -30502.229} C_VEL
LIN {X 0,Y 26.119,Z 505.757,A -85,B 0,C 180,E1 -30515.793,E2 -30515.793} C_VEL
LIN {X 0,Y 21.519,Z 513.424,A -85,B 0,C 180,E1 -30536.086,E2 -30536.086} C_VEL
LIN {X 0,Y 20.185,Z 519.708,A -85,B 0,C 180,E1 -30562.453,E2 -30562.453} C_VEL
LIN {X 0,Y 24.128,Z 526.033,A -85,B 0,C 180,E1 -30592.213,E2 -30592.213} C_VEL
LIN {X 0,Y 33.309,Z 531.459,A -85,B 0,C 180,E1 -30612.178,E2 -30612.178} C_VEL
LIN {X 0,Y 42.541,Z 534.818,A -85,B 0,C 180,E1 -30621.365,E2 -30621.365} C_VEL
LIN {X 0,Y 40.491,Z 534.358,A -85,B 0,C 180,E1 -30624.734,E2 -30624.734} C_VEL
LIN {X 0,Y 30.853,Z 530.997,A -85,B 0,C 180,E1 -30637.119,E2 -30637.119} C_VEL
LIN {X 0,Y 23.302,Z 525.708,A -85,B 0,C 180,E1 -30663.1,E2 -30663.1} C_VEL
LIN {X 0,Y 21.978,Z 522.713,A -85,B 0,C 180,E1 -30678.88,E2 -30678.88} C_VEL
LIN {X 0,Y 21.722,Z 516.957,A -85,B 0,C 180,E1 -30703.933,E2 -30703.933} C_VEL
LIN {X 0,Y 25.424,Z 508.883,A -85,B 0,C 180,E1 -30728.448,E2 -30728.448} C_VEL
LIN {X 0,Y 30.99,Z 500.644,A -85,B 0,C 180,E1 -30742.524,E2 -30742.524} C_VEL
LIN {X 0,Y 37.8,Z 490.522,A -85,B 0,C 180,E1 -30752.011,E2 -30752.011} C_VEL
LIN {X 0,Y 44.522,Z 479.231,A -85,B 0,C 180,E1 -30758.016,E2 -30758.016} C_VEL
LIN {X 0,Y 50.018,Z 468.272,A -85,B 0,C 180,E1 -30761.505,E2 -30761.505} C_VEL
LIN {X 0,Y 55.254,Z 454.979,A -85,B 0,C 180,E1 -30764.116,E2 -30764.116} C_VEL
LIN {X 0,Y 58.983,Z 442.07,A -85,B 0,C 180,E1 -30765.698,E2 -30765.698} C_VEL
LIN {X 0,Y 61.562,Z 427.918,A -85,B 0,C 180,E1 -30766.803,E2 -30766.803} C_VEL
LIN {X 0,Y 64.287,Z 409.728,A -85,B 0,C 180,E1 -30767.961,E2 -30767.961} C_VEL
LIN {X 0,Y 63.31,Z 403.329,A -85,B 0,C 180,E1 -30771.199,E2 -30771.199} C_VEL
LIN {X 0,Y 61.467,Z 396.726,A -85,B 0,C 180,E1 -30776.494,E2 -30776.494} C_VEL
LIN {X 0,Y 59.77,Z 391.313,A -85,B 0,C 180,E1 -30782.608,E2 -30782.608} C_VEL
LIN {X 0,Y 58.656,Z 387.669,A -85,B 0,C 180,E1 -30788.169,E2 -30788.169} C_VEL
LIN {X 0,Y 58.167,Z 386.164,A -85,B 0,C 180,E1 -30791.174,E2 -30791.174} C_VEL
LIN {X 0,Y 57.461,Z 384.103,A -85,B 0,C 180,E1 -30797.913,E2 -30797.913} C_VEL
LIN {X 0,Y 57.281,Z 384.412,A -85,B 0,C 180,E1 -30807.987,E2 -30807.987} C_VEL
LIN {X 0,Y 58.368,Z 388.051,A -85,B 0,C 180,E1 -30818.868,E2 -30818.868} C_VEL
LIN {X 0,Y 59.834,Z 391.665,A -85,B 0,C 180,E1 -30825.475,E2 -30825.475} C_VEL
LIN {X 0,Y 62.137,Z 398.104,A -85,B 0,C 180,E1 -30833.056,E2 -30833.056} C_VEL
LIN {X 0,Y 63.99,Z 404.296,A -85,B 0,C 180,E1 -30837.925,E2 -30837.925} C_VEL
LIN {X 0,Y 64.49,Z 406.614,A -85,B 0,C 180,E1 -30839.257,E2 -30839.257} C_VEL
LIN {X 0,Y 59.979,Z 434.674,A -85,B 0,C 180,E1 -30840.922,E2 -30840.922} C_VEL
LIN {X 0,Y 56.858,Z 447.419,A -85,B 0,C 180,E1 -30842.322,E2 -30842.322} C_VEL
LIN {X 0,Y 52.82,Z 459.311,A -85,B 0,C 180,E1 -30844.296,E2 -30844.296} C_VEL
LIN {X 0,Y 51.408,Z 462.819,A -85,B 0,C 180,E1 -30845.06,E2 -30845.06} C_VEL
LIN {X 0,Y 48.684,Z 468.062,A -85,B 0,C 180,E1 -30845.761,E2 -30845.761} C_VEL
LIN {X 0,Y 42.842,Z 476.06,A -85,B 0,C 180,E1 -30845.419,E2 -30845.419} C_VEL
LIN {X 0,Y 36.469,Z 483.737,A -85,B 0,C 180,E1 -30845.266,E2 -30845.266} C_VEL
LIN {X 0,Y 32.927,Z 488.384,A -85,B 0,C 180,E1 -30846.877,E2 -30846.877} C_VEL
LIN {X 0,Y 25.191,Z 498.776,A -85,B 0,C 180,E1 -30855.794,E2 -30855.794} C_VEL
LIN {X 0,Y 18.094,Z 507.66,A -85,B 0,C 180,E1 -30872.796,E2 -30872.796} C_VEL
LIN {X 0,Y 13.726,Z 514.425,A -85,B 0,C 180,E1 -30900.818,E2 -30900.818} C_VEL
LIN {X 0,Y 14.621,Z 521.049,A -85,B 0,C 180,E1 -30944.08,E2 -30944.08} C_VEL
LIN {X 0,Y 21.509,Z 526.595,A -85,B 0,C 180,E1 -30971.354,E2 -30971.354} C_VEL
LIN {X 0,Y 28.487,Z 530.084,A -85,B 0,C 180,E1 -30981.923,E2 -30981.923} C_VEL
LIN {X 0,Y 27.106,Z 529.565,A -85,B 0,C 180,E1 -30985.489,E2 -30985.489} C_VEL
LIN {X 0,Y 18.027,Z 524.551,A -85,B 0,C 180,E1 -31009.422,E2 -31009.422} C_VEL
LIN {X 0,Y 15.074,Z 520.462,A -85,B 0,C 180,E1 -31036.504,E2 -31036.504} C_VEL
LIN {X 0,Y 15.162,Z 514.5,A -85,B 0,C 180,E1 -31072.037,E2 -31072.037} C_VEL
LIN {X 0,Y 20.416,Z 506.274,A -85,B 0,C 180,E1 -31100.745,E2 -31100.745} C_VEL
LIN {X 0,Y 27.309,Z 497.544,A -85,B 0,C 180,E1 -31114.235,E2 -31114.235} C_VEL
LIN {X 0,Y 35.064,Z 486.801,A -85,B 0,C 180,E1 -31122.166,E2 -31122.166} C_VEL
LIN {X 0,Y 42.411,Z 474.583,A -85,B 0,C 180,E1 -31126.769,E2 -31126.769} C_VEL
LIN {X 0,Y 48.265,Z 462.428,A -85,B 0,C 180,E1 -31129.359,E2 -31129.359} C_VEL
LIN {X 0,Y 53.353,Z 448.438,A -85,B 0,C 180,E1 -31131.062,E2 -31131.062} C_VEL
LIN {X 0,Y 56.54,Z 435.477,A -85,B 0,C 180,E1 -31132.126,E2 -31132.126} C_VEL
LIN {X 0,Y 60.414,Z 411.114,A -85,B 0,C 180,E1 -31133.545,E2 -31133.545} C_VEL
LIN {X 0,Y 59.838,Z 406.823,A -85,B 0,C 180,E1 -31136.093,E2 -31136.093} C_VEL
LIN {X 0,Y 58.589,Z 401.147,A -85,B 0,C 180,E1 -31141.191,E2 -31141.191} C_VEL
LIN {X 0,Y 57.464,Z 396.317,A -85,B 0,C 180,E1 -31147.202,E2 -31147.202} C_VEL
LIN {X 0,Y 56.699,Z 392.857,A -85,B 0,C 180,E1 -31152.969,E2 -31152.969} C_VEL
LIN {X 0,Y 56.258,Z 391.245,A -85,B 0,C 180,E1 -31158.31,E2 -31158.31} C_VEL
LIN {X 0,Y 56.098,Z 391.223,A -85,B 0,C 180,E1 -31166.208,E2 -31166.208} C_VEL
LIN {X 0,Y 56.759,Z 394.694,A -85,B 0,C 180,E1 -31176.752,E2 -31176.752} C_VEL
LIN {X 0,Y 57.843,Z 397.976,A -85,B 0,C 180,E1 -31182.836,E2 -31182.836} C_VEL
LIN {X 0,Y 59.452,Z 403.777,A -85,B 0,C 180,E1 -31189.746,E2 -31189.746} C_VEL
LIN {X 0,Y 60.595,Z 408.685,A -85,B 0,C 180,E1 -31193.792,E2 -31193.792} C_VEL
LIN {X 0,Y 56.06,Z 435.49,A -85,B 0,C 180,E1 -31195.017,E2 -31195.017} C_VEL
LIN {X 0,Y 52.431,Z 449.361,A -85,B 0,C 180,E1 -31196.346,E2 -31196.346} C_VEL
LIN {X 0,Y 47.632,Z 462.137,A -85,B 0,C 180,E1 -31198.161,E2 -31198.161} C_VEL
LIN {X 0,Y 41.243,Z 475.131,A -85,B 0,C 180,E1 -31201.236,E2 -31201.236} C_VEL
LIN {X 0,Y 34.263,Z 486.463,A -85,B 0,C 180,E1 -31205.788,E2 -31205.788} C_VEL
LIN {X 0,Y 32.927,Z 488.384,A -85,B 0,C 180,E1 -31206.877,E2 -31206.877} C_VEL
LIN {X 0,Y 29.276,Z 492.88,A -85,B 0,C 180,E1 -31209.009,E2 -31209.009} C_VEL
LIN {X 0,Y 21.996,Z 499.547,A -85,B 0,C 180,E1 -31210.864,E2 -31210.864} C_VEL
LIN {X 0,Y 15.761,Z 504.494,A -85,B 0,C 180,E1 -31213.466,E2 -31213.466} C_VEL
LIN {X 0,Y 11.368,Z 508.213,A -85,B 0,C 180,E1 -31220.446,E2 -31220.446} C_VEL
LIN {X 0,Y 10.097,Z 509.447,A -85,B 0,C 180,E1 -31225.149,E2 -31225.149} C_VEL
LIN {X 0,Y 6.637,Z 516.981,A -85,B 0,C 180,E1 -31298.628,E2 -31298.628} C_VEL
LIN {X 0,Y 13.87,Z 522.961,A -85,B 0,C 180,E1 -31342.329,E2 -31342.329} C_VEL
LIN {X 0,Y 12.669,Z 522.223,A -85,B 0,C 180,E1 -31353.683,E2 -31353.683} C_VEL
LIN {X 0,Y 8.535,Z 518.473,A -85,B 0,C 180,E1 -31385.658,E2 -31385.658} C_VEL
LIN {X 0,Y 9.87,Z 511.091,A -85,B 0,C 180,E1 -31455.367,E2 -31455.367} C_VEL
LIN {X 0,Y 18.496,Z 501.788,A -85,B 0,C 180,E1 -31481.749,E2 -31481.749} C_VEL
LIN {X 0,Y 26.756,Z 492.173,A -85,B 0,C 180,E1 -31490.01,E2 -31490.01} C_VEL
LIN {X 0,Y 34.451,Z 481.492,A -85,B 0,C 180,E1 -31493.914,E2 -31493.914} C_VEL
LIN {X 0,Y 41.376,Z 469.512,A -85,B 0,C 180,E1 -31496.198,E2 -31496.198} C_VEL
LIN {X 0,Y 47.039,Z 456.962,A -85,B 0,C 180,E1 -31497.522,E2 -31497.522} C_VEL
LIN {X 0,Y 51.489,Z 443.418,A -85,B 0,C 180,E1 -31498.365,E2 -31498.365} C_VEL
LIN {X 0,Y 54.118,Z 431.376,A -85,B 0,C 180,E1 -31498.952,E2 -31498.952} C_VEL
LIN {X 0,Y 57.123,Z 412.762,A -85,B 0,C 180,E1 -31499.733,E2 -31499.733} C_VEL
LIN {X 0,Y 56.455,Z 407.451,A -85,B 0,C 180,E1 -31504.172,E2 -31504.172} C_VEL
LIN {X 0,Y 55.613,Z 402.505,A -85,B 0,C 180,E1 -31510.343,E2 -31510.343} C_VEL
LIN {X 0,Y 55.218,Z 399.393,A -85,B 0,C 180,E1 -31515.511,E2 -31515.511} C_VEL
LIN {X 0,Y 54.986,Z 398.164,A -85,B 0,C 180,E1 -31520.334,E2 -31520.334} C_VEL
LIN {X 0,Y 54.915,Z 398.33,A -85,B 0,C 180,E1 -31525.231,E2 -31525.231} C_VEL
LIN {X 0,Y 55.225,Z 401.297,A -85,B 0,C 180,E1 -31534.451,E2 -31534.451} C_VEL
LIN {X 0,Y 55.874,Z 404.146,A -85,B 0,C 180,E1 -31539.747,E2 -31539.747} C_VEL
LIN {X 0,Y 56.974,Z 409.327,A -85,B 0,C 180,E1 -31546.052,E2 -31546.052} C_VEL
LIN {X 0,Y 57.217,Z 411.336,A -85,B 0,C 180,E1 -31547.63,E2 -31547.63} C_VEL
LIN {X 0,Y 52.942,Z 435.757,A -85,B 0,C 180,E1 -31548.271,E2 -31548.271} C_VEL
LIN {X 0,Y 49.241,Z 449.471,A -85,B 0,C 180,E1 -31549.18,E2 -31549.18} C_VEL
LIN {X 0,Y 44.065,Z 462.722,A -85,B 0,C 180,E1 -31550.366,E2 -31550.366} C_VEL
LIN {X 0,Y 37.403,Z 475.565,A -85,B 0,C 180,E1 -31552.37,E2 -31552.37} C_VEL
LIN {X 0,Y 30.631,Z 485.93,A -85,B 0,C 180,E1 -31555.008,E2 -31555.008} C_VEL
LIN {X 0,Y 22.39,Z 496.339,A -85,B 0,C 180,E1 -31560.374,E2 -31560.374} C_VEL
LIN {X 0,Y 13.907,Z 505.539,A -85,B 0,C 180,E1 -31572.651,E2 -31572.651} C_VEL
LIN {X 0,Y 10.097,Z 509.447,A -85,B 0,C 180,E1 -31585.149,E2 -31585.149} C_VEL
LIN {X 0,Y 8.758,Z 509.945,A -85,B 0,C 180,E1 -31584.093,E2 -31584.093} C_VEL
LIN {X 0,Y 7.045,Z 509.539,A -85,B 0,C 180,E1 -31568.918,E2 -31568.918} C_VEL
LIN {X 0,Y 7.128,Z 508.076,A -85,B 0,C 180,E1 -31541.14,E2 -31541.14} C_VEL
LIN {X 0,Y 8.811,Z 506.305,A -85,B 0,C 180,E1 -31524.316,E2 -31524.316} C_VEL
LIN {X 0,Y 16.665,Z 499.285,A -85,B 0,C 180,E1 -31507.185,E2 -31507.185} C_VEL
LIN {X 0,Y 20.595,Z 495.35,A -85,B 0,C 180,E1 -31505.114,E2 -31505.114} C_VEL
LIN {X 0,Y 24.276,Z 491.134,A -85,B 0,C 180,E1 -31504.776,E2 -31504.776} C_VEL
LIN {X 0,Y 31.758,Z 481.025,A -85,B 0,C 180,E1 -31505.315,E2 -31505.315} C_VEL
LIN {X 0,Y 38.84,Z 469.096,A -85,B 0,C 180,E1 -31505.677,E2 -31505.677} C_VEL
LIN {X 0,Y 44.593,Z 456.579,A -85,B 0,C 180,E1 -31505.863,E2 -31505.863} C_VEL
LIN {X 0,Y 49.151,Z 442.932,A -85,B 0,C 180,E1 -31505.978,E2 -31505.978} C_VEL
LIN {X 0,Y 51.914,Z 430.337,A -85,B 0,C 180,E1 -31506.227,E2 -31506.227} C_VEL
LIN {X 0,Y 54.464,Z 414.906,A -85,B 0,C 180,E1 -31506.584,E2 -31506.584} C_VEL
LIN {X 0,Y 54.07,Z 410.211,A -85,B 0,C 180,E1 -31511.536,E2 -31511.536} C_VEL
LIN {X 0,Y 53.849,Z 405.871,A -85,B 0,C 180,E1 -31518.343,E2 -31518.343} C_VEL
LIN {X 0,Y 53.809,Z 405.208,A -85,B 0,C 180,E1 -31520.8,E2 -31520.8} C_VEL
LIN {X 0,Y 53.75,Z 405.269,A -85,B 0,C 180,E1 -31523.768,E2 -31523.768} C_VEL
LIN {X 0,Y 53.794,Z 407.934,A -85,B 0,C 180,E1 -31532.158,E2 -31532.158} C_VEL
LIN {X 0,Y 54.077,Z 410.253,A -85,B 0,C 180,E1 -31536.376,E2 -31536.376} C_VEL
LIN {X 0,Y 54.518,Z 413.589,A -85,B 0,C 180,E1 -31540.684,E2 -31540.684} C_VEL
LIN {X 0,Y 50.908,Z 434.356,A -85,B 0,C 180,E1 -31540.869,E2 -31540.869} C_VEL
LIN {X 0,Y 47.468,Z 447.437,A -85,B 0,C 180,E1 -31541.12,E2 -31541.12} C_VEL
LIN {X 0,Y 42.52,Z 460.579,A -85,B 0,C 180,E1 -31541.391,E2 -31541.391} C_VEL
LIN {X 0,Y 36.538,Z 472.53,A -85,B 0,C 180,E1 -31541.648,E2 -31541.648} C_VEL
LIN {X 0,Y 29.466,Z 483.662,A -85,B 0,C 180,E1 -31541.97,E2 -31541.97} C_VEL
LIN {X 0,Y 20.871,Z 494.6,A -85,B 0,C 180,E1 -31542.343,E2 -31542.343} C_VEL
LIN {X 0,Y 12.392,Z 503.417,A -85,B 0,C 180,E1 -31542.659,E2 -31542.659} C_VEL
LIN {X 0,Y 5.066,Z 509.745,A -85,B 0,C 180,E1 -31539.248,E2 -31539.248} C_VEL
LIN {X 0,Y 0.922,Z 513.077,A -85,B 0,C 180,E1 -31500.104,E2 -31500.104} C_VEL
LIN {X 0,Y 2.862,Z 511.865,A -85,B 0,C 180,E1 -31491.691,E2 -31491.691} C_VEL
LIN {X 0,Y 12.31,Z 503.886,A -85,B 0,C 180,E1 -31502.852,E2 -31502.852} C_VEL
LIN {X 0,Y 22.026,Z 493.794,A -85,B 0,C 180,E1 -31504.489,E2 -31504.489} C_VEL
LIN {X 0,Y 24.276,Z 491.134,A -85,B 0,C 180,E1 -31504.776,E2 -31504.776} C_VEL
LIN {X 0,Y 27.722,Z 486.451,A -85,B 0,C 180,E1 -31506.407,E2 -31506.407} C_VEL
LIN {X 0,Y 32.59,Z 478.239,A -85,B 0,C 180,E1 -31511.447,E2 -31511.447} C_VEL
LIN {X 0,Y 37.044,Z 469.621,A -85,B 0,C 180,E1 -31515.251,E2 -31515.251} C_VEL
LIN {X 0,Y 39.642,Z 464.193,A -85,B 0,C 180,E1 -31515.577,E2 -31515.577} C_VEL
LIN {X 0,Y 44.699,Z 451.919,A -85,B 0,C 180,E1 -31514.627,E2 -31514.627} C_VEL
LIN {X 0,Y 48.532,Z 438.893,A -85,B 0,C 180,E1 -31514.037,E2 -31514.037} C_VEL
LIN {X 0,Y 52.447,Z 417.501,A -85,B 0,C 180,E1 -31513.866,E2 -31513.866} C_VEL
LIN {X 0,Y 52.53,Z 413.413,A -85,B 0,C 180,E1 -31519.45,E2 -31519.45} C_VEL
LIN {X 0,Y 52.593,Z 412.631,A -85,B 0,C 180,E1 -31520.72,E2 -31520.72} C_VEL
LIN {X 0,Y 52.524,Z 412.787,A -85,B 0,C 180,E1 -31524.359,E2 -31524.359} C_VEL
LIN {X 0,Y 52.46,Z 414.74,A -85,B 0,C 180,E1 -31530.164,E2 -31530.164} C_VEL
LIN {X 0,Y 52.485,Z 416.705,A -85,B 0,C 180,E1 -31533.27,E2 -31533.27} C_VEL
LIN {X 0,Y 49.396,Z 434.4,A -85,B 0,C 180,E1 -31532.888,E2 -31532.888} C_VEL
LIN {X 0,Y 46.173,Z 446.931,A -85,B 0,C 180,E1 -31532.612,E2 -31532.612} C_VEL
LIN {X 0,Y 41.362,Z 459.979,A -85,B 0,C 180,E1 -31531.847,E2 -31531.847} C_VEL
LIN {X 0,Y 35.595,Z 471.882,A -85,B 0,C 180,E1 -31530.501,E2 -31530.501} C_VEL
LIN {X 0,Y 28.721,Z 483.087,A -85,B 0,C 180,E1 -31528.077,E2 -31528.077} C_VEL
LIN {X 0,Y 23.231,Z 490.632,A -85,B 0,C 180,E1 -31524.854,E2 -31524.854} C_VEL
LIN {X 0,Y 22.752,Z 491.277,A -85,B 0,C 180,E1 -31522.105,E2 -31522.105} C_VEL
LIN {X 0,Y 30.517,Z 480.525,A -85,B 0,C 180,E1 -31518.222,E2 -31518.222} C_VEL
LIN {X 0,Y 37.489,Z 468.57,A -85,B 0,C 180,E1 -31516.126,E2 -31516.126} C_VEL
LIN {X 0,Y 39.642,Z 464.193,A -85,B 0,C 180,E1 -31515.577,E2 -31515.577} C_VEL
LIN {X 0,Y 41.991,Z 458.78,A -85,B 0,C 180,E1 -31515.911,E2 -31515.911} C_VEL
LIN {X 0,Y 45.134,Z 449.636,A -85,B 0,C 180,E1 -31518.831,E2 -31518.831} C_VEL
LIN {X 0,Y 47.65,Z 440.243,A -85,B 0,C 180,E1 -31521.694,E2 -31521.694} C_VEL
LIN {X 0,Y 48.875,Z 434.423,A -85,B 0,C 180,E1 -31522.177,E2 -31522.177} C_VEL
LIN {X 0,Y 51.276,Z 420.416,A -85,B 0,C 180,E1 -31521.871,E2 -31521.871} C_VEL
LIN {X 0,Y 51.326,Z 420.052,A -85,B 0,C 180,E1 -31524.096,E2 -31524.096} C_VEL
LIN {X 0,Y 51.249,Z 420.685,A -85,B 0,C 180,E1 -31525.446,E2 -31525.446} C_VEL
LIN {X 0,Y 47.889,Z 438.888,A -85,B 0,C 180,E1 -31524.351,E2 -31524.351} C_VEL
LIN {X 0,Y 45.572,Z 447.467,A -85,B 0,C 180,E1 -31523.7,E2 -31523.7} C_VEL
LIN {X 0,Y 46.116,Z 445.677,A -85,B 0,C 180,E1 -31523.014,E2 -31523.014} C_VEL
LIN {X 0,Y 48.875,Z 434.423,A -85,B 0,C 180,E1 -31522.177,E2 -31522.177} C_VEL
LIN {X 0,Y 52.774,Z 434.797,A -85,B 0,C 180,E1 -31521.363,E2 -31521.363} C_VEL
LIN {X 0,Y 52.774,Z 600,A -85,B 0,C 180,E1 -31521.363,E2 -31521.363} C_VEL
LIN {X 0,Y 52.774,Z 600,A -85,B 0,C 180,E1 -31521.363,E2 -31521.363}

QRS_NEXT_CUT()

QRS_NEXT()
QRS_HOME()

END
